(* IEC 61131-3 sources: SmartHomeNew/ (part 13) *)

(* ---- PRG_IO_Read_Phase_03_Environment_Sensors.st ---- *)
PROGRAM PRG_IO_Read_Phase_03_Environment_Sensors
VAR
    L_i : INT;
    L_Filtered_Room_Temp : REAL;
    L_Filtered_Floor_Temp : REAL;
    L_Any_Sensor_Fault : BOOL;

    fbCalib_Outdoor_Temp : FB_Sensor_Calibration_Processor;
    fbCalib_Supply_Temps : ARRAY[1..GVL_CONSTANTS.C_MAX_SUPPLY_TEMPS] OF FB_Sensor_Calibration_Processor;
    fbCalib_Room_Temps : ARRAY[1..GVL_CONSTANTS.C_MAX_ZONES] OF FB_Sensor_Calibration_Processor;
    fbCalib_Floor_Temps : ARRAY[1..GVL_CONSTANTS.C_MAX_ZONES] OF FB_Sensor_Calibration_Processor;
    fbCalib_Room_Hum : ARRAY[1..GVL_CONSTANTS.C_MAX_ZONES] OF FB_Sensor_Calibration_Processor;
    fbCalib_Room_CO2 : ARRAY[1..GVL_CONSTANTS.C_MAX_ZONES] OF FB_Sensor_Calibration_Processor;
END_VAR

L_Any_Sensor_Fault := FALSE;

fbCalib_Outdoor_Temp(
    VI_Raw_Value := GVL_IO.AI_Temp_Outdoor.rValue,
    VI_Record := GVL_CONFIG.G_Calib_Outdoor_Temp
);
GVL_STATE.G_Outdoor_Temp := fbCalib_Outdoor_Temp.VO_Calibrated_Value;

FOR L_i := 1 TO GVL_CONSTANTS.C_MAX_SUPPLY_TEMPS DO
    IF GVL_IO.AI_Supply_Temps[L_i].wStatus = 0 THEN
        fbCalib_Supply_Temps[L_i](
            VI_Raw_Value := GVL_IO.AI_Supply_Temps[L_i].rValue,
            VI_Record := GVL_CONFIG.G_Calib_Supply_Temps[L_i]
        );
        GVL_STATE.G_Supply_Temps[L_i] := fbCalib_Supply_Temps[L_i].VO_Calibrated_Value;
    ELSE
        L_Any_Sensor_Fault := TRUE;
    END_IF;
END_FOR;

FOR L_i := 1 TO GVL_CONSTANTS.C_MAX_ZONES DO
    fbCalib_Room_Hum[L_i](
        VI_Raw_Value := GVL_IO.AI_Room_Hum[L_i],
        VI_Record := GVL_CONFIG.G_Calib_Humidity[L_i]
    );
    GVL_STATE.G_Room_Hum[L_i] := fbCalib_Room_Hum[L_i].VO_Calibrated_Value;

    fbCalib_Room_CO2[L_i](
        VI_Raw_Value := GVL_IO.AI_Room_CO2[L_i],
        VI_Record := GVL_CONFIG.G_Calib_CO2[L_i]
    );
    GVL_STATE.G_Room_CO2[L_i] := fbCalib_Room_CO2[L_i].VO_Calibrated_Value;
END_FOR;

FOR L_i := 1 TO GVL_CONSTANTS.C_MAX_ZONES DO
    fbCalib_Room_Temps[L_i](
        VI_Raw_Value := GVL_IO.AI_Room_Temps[L_i],
        VI_Record := GVL_CONFIG.G_Calib_Room_Temps[L_i]
    );

    IF GVL_STATE.G_Last_Valid_Room_Temps[L_i] = 0.0 THEN
        L_Filtered_Room_Temp := fbCalib_Room_Temps[L_i].VO_Calibrated_Value;
    ELSE
        L_Filtered_Room_Temp := (GVL_STATE.G_Last_Valid_Room_Temps[L_i] * 0.9) + (fbCalib_Room_Temps[L_i].VO_Calibrated_Value * 0.1);
    END_IF;

    IF (L_Filtered_Room_Temp < -50.0) OR (L_Filtered_Room_Temp > 100.0) THEN
        GVL_STATE.G_Temp_Sensor_Fault[L_i] := TRUE;
        GVL_STATE.G_Room_Temps[L_i] := GVL_STATE.G_Last_Valid_Room_Temps[L_i];
        L_Any_Sensor_Fault := TRUE;
    ELSE
        GVL_STATE.G_Temp_Sensor_Fault[L_i] := FALSE;
        GVL_STATE.G_Room_Temps[L_i] := L_Filtered_Room_Temp;
        GVL_STATE.G_Last_Valid_Room_Temps[L_i] := L_Filtered_Room_Temp;
    END_IF;
END_FOR;

FOR L_i := 1 TO GVL_CONSTANTS.C_MAX_HEATING_CIRCUITS DO
    IF L_i <= GVL_CONSTANTS.C_MAX_ZONES THEN
        fbCalib_Floor_Temps[L_i](
            VI_Raw_Value := GVL_IO.AI_Floor_Temps[L_i],
            VI_Record := GVL_CONFIG.G_Calib_Floor_Temps[L_i]
        );

        IF GVL_STATE.G_Last_Valid_Floor_Temps[L_i] = 0.0 THEN
            L_Filtered_Floor_Temp := fbCalib_Floor_Temps[L_i].VO_Calibrated_Value;
        ELSE
            L_Filtered_Floor_Temp := (GVL_STATE.G_Last_Valid_Floor_Temps[L_i] * 0.9) + (fbCalib_Floor_Temps[L_i].VO_Calibrated_Value * 0.1);
        END_IF;

        IF (L_Filtered_Floor_Temp < -50.0) OR (L_Filtered_Floor_Temp > 100.0) THEN
            GVL_STATE.G_Floor_Temp_Sensor_Fault[L_i] := TRUE;
            GVL_STATE.G_Floor_Temps[L_i] := GVL_STATE.G_Last_Valid_Floor_Temps[L_i];
            L_Any_Sensor_Fault := TRUE;
        ELSE
            GVL_STATE.G_Floor_Temp_Sensor_Fault[L_i] := FALSE;
            GVL_STATE.G_Floor_Temps[L_i] := L_Filtered_Floor_Temp;
            GVL_STATE.G_Last_Valid_Floor_Temps[L_i] := L_Filtered_Floor_Temp;
        END_IF;
    ELSE
        GVL_STATE.G_Floor_Temp_Sensor_Fault[L_i] := TRUE;
        GVL_STATE.G_Floor_Temps[L_i] := GVL_STATE.G_Last_Valid_Floor_Temps[L_i];
        L_Any_Sensor_Fault := TRUE;
    END_IF;
END_FOR;

GVL_STATUS.G_Diagnostics.Sensor_Fault := L_Any_Sensor_Fault;

// >>> BULK_SYNC_ANCHOR: PRG_IO_Read_Phase_03_Environment_Sensors <<<
END_PROGRAM

(* ---- PRG_IO_Read_Phase_04_Heating_Manifold_Sensors.st ---- *)
PROGRAM PRG_IO_Read_Phase_04_Heating_Manifold_Sensors
VAR
    L_i : INT;
    L_Manifold_Pressure_Raw : WORD;
    L_Manifold_Current_Raw : WORD;

    fbDiagEventManager : FB_Diagnostics_Event_Manager;
    fbCalib_Manifold_T_Supply : ARRAY[1..GVL_CONSTANTS.C_MAX_MANIFOLDS] OF FB_Sensor_Calibration_Processor;
    fbCalib_Manifold_T_Return : ARRAY[1..GVL_CONSTANTS.C_MAX_MANIFOLDS] OF FB_Sensor_Calibration_Processor;
    fbAnalog_Manifold_Pressure : ARRAY[1..GVL_CONSTANTS.C_MAX_MANIFOLDS] OF FB_Sensor_Analog_Processing;
    fbAnalog_Manifold_Current : ARRAY[1..GVL_CONSTANTS.C_MAX_MANIFOLDS] OF FB_Sensor_Analog_Processing;
END_VAR

GVL_STATUS.G_Diagnostics.Manifold_Pressure_Fault_Active := FALSE;
GVL_STATUS.G_Diagnostics.Manifold_Pressure_First_Fault_Index := 0;
GVL_STATUS.G_Diagnostics.Manifold_Current_Fault_Active := FALSE;
GVL_STATUS.G_Diagnostics.Manifold_Current_First_Fault_Index := 0;
GVL_STATUS.G_Diagnostics.Manifold_Pressure_Fault_Text := '';
GVL_STATUS.G_Diagnostics.Manifold_Current_Fault_Text := '';

FOR L_i := 1 TO GVL_CONSTANTS.C_MAX_MANIFOLDS DO
    IF GVL_IO.AI_Manifold_Pressures[L_i] < 0 THEN
        L_Manifold_Pressure_Raw := 0;
    ELSE
        L_Manifold_Pressure_Raw := INT_TO_WORD(GVL_IO.AI_Manifold_Pressures[L_i]);
    END_IF;

    IF GVL_IO.AI_Manifold_Currents[L_i] < 0 THEN
        L_Manifold_Current_Raw := 0;
    ELSE
        L_Manifold_Current_Raw := INT_TO_WORD(GVL_IO.AI_Manifold_Currents[L_i]);
    END_IF;

    fbAnalog_Manifold_Pressure[L_i](
        VI_Raw_Value := L_Manifold_Pressure_Raw,
        VI_Sensor_Type := 0,
        VI_Min_Scale := 0.0,
        VI_Max_Scale := 10.0,
        VI_Offset := 0.0,
        VI_Multiplier := 1.0,
        VI_Filter_Time_MS := GVL_CONSTANTS.C_MS_IN_SECOND,
        VI_System_Time_MS := GVL_STATUS.G_System_Time_MS,
        VI_Fallback_Mode := 0,
        VI_Default_Value := 0.0
    );
    GVL_STATE.G_Manifold_Pressures[L_i] := fbAnalog_Manifold_Pressure[L_i].VO_Value;
    GVL_STATUS.G_Diagnostics.Manifold_Pressure_Fault[L_i] := fbAnalog_Manifold_Pressure[L_i].VO_Error;
    GVL_STATUS.G_Diagnostics.Manifold_Pressure_Diag_Code[L_i] := fbAnalog_Manifold_Pressure[L_i].VO_Diag_Code;

    fbDiagEventManager(
        VI_Code := GVL_CONFIG.ERR_PRESSURE_OUT_OF_RANGE,
        VI_Severity := 3,
        VI_Active := fbAnalog_Manifold_Pressure[L_i].VO_Error,
        VI_Timestamp := GVL_STATUS.G_System_Time_MS,
        VI_Source := 100 + L_i,
        VIO_Events := GVL_STATUS.G_Diagnostics_Events,
        VIO_Count := GVL_STATUS.G_Diagnostics_Count
    );

    fbAnalog_Manifold_Current[L_i](
        VI_Raw_Value := L_Manifold_Current_Raw,
        VI_Sensor_Type := 0,
        VI_Min_Scale := 0.0,
        VI_Max_Scale := 16.0,
        VI_Offset := 0.0,
        VI_Multiplier := 1.0,
        VI_Filter_Time_MS := GVL_CONSTANTS.C_MS_IN_SECOND,
        VI_System_Time_MS := GVL_STATUS.G_System_Time_MS,
        VI_Fallback_Mode := 0,
        VI_Default_Value := 0.0
    );
    GVL_STATE.G_Manifold_Currents[L_i] := fbAnalog_Manifold_Current[L_i].VO_Value;
    GVL_STATUS.G_Diagnostics.Manifold_Current_Fault[L_i] := fbAnalog_Manifold_Current[L_i].VO_Error;
    GVL_STATUS.G_Diagnostics.Manifold_Current_Diag_Code[L_i] := fbAnalog_Manifold_Current[L_i].VO_Diag_Code;

    fbDiagEventManager(
        VI_Code := GVL_CONFIG.ERR_PUMP_UNDERCURRENT,
        VI_Severity := 3,
        VI_Active := fbAnalog_Manifold_Current[L_i].VO_Error,
        VI_Timestamp := GVL_STATUS.G_System_Time_MS,
        VI_Source := 200 + L_i,
        VIO_Events := GVL_STATUS.G_Diagnostics_Events,
        VIO_Count := GVL_STATUS.G_Diagnostics_Count
    );

    IF GVL_IO.AI_Manifold_Temps_Supply[L_i].wStatus = 0 THEN
        fbCalib_Manifold_T_Supply[L_i](
            VI_Raw_Value := GVL_IO.AI_Manifold_Temps_Supply[L_i].rValue,
            VI_Record := GVL_CONFIG.G_Calib_Manifold_T_Supply[L_i]
        );
        GVL_STATE.G_Manifold_T_Supply[L_i] := fbCalib_Manifold_T_Supply[L_i].VO_Calibrated_Value;
    END_IF;

    fbCalib_Manifold_T_Return[L_i](
        VI_Raw_Value := INT_TO_REAL(GVL_IO.AI_Manifold_Temps_Return[L_i]) / 10.0,
        VI_Record := GVL_CONFIG.G_Calib_Manifold_T_Return[L_i]
    );
    GVL_STATE.G_Manifold_T_Return[L_i] := fbCalib_Manifold_T_Return[L_i].VO_Calibrated_Value;
    GVL_STATE.G_Manifold_End_Switches[L_i] := GVL_IO.DI_Manifold_End_Switches[L_i];

    IF GVL_STATUS.G_Diagnostics.Manifold_Pressure_Fault[L_i] OR GVL_STATUS.G_Diagnostics.Manifold_Current_Fault[L_i] THEN
        GVL_STATUS.G_Diagnostics.Sensor_Fault := TRUE;
        GVL_STATUS.G_Diagnostics.Subsystem_Degraded := TRUE;
    END_IF;

    IF GVL_STATUS.G_Diagnostics.Manifold_Pressure_Fault[L_i] AND GVL_STATUS.G_Diagnostics.Manifold_Current_Fault[L_i] THEN
        GVL_STATUS.G_Diagnostics.Manifold_Pressure_Fault_Text := 'Correlated pressure/current fault detected';
        GVL_STATUS.G_Diagnostics.Manifold_Current_Fault_Text := 'Correlated pressure/current fault detected';
    ELSIF GVL_STATUS.G_Diagnostics.Manifold_Pressure_Fault[L_i] AND (GVL_STATUS.G_Diagnostics.Manifold_Pressure_Fault_Text = '') THEN
        GVL_STATUS.G_Diagnostics.Manifold_Pressure_Fault_Text := 'Pressure sensor fault detected';
    ELSIF GVL_STATUS.G_Diagnostics.Manifold_Current_Fault[L_i] AND (GVL_STATUS.G_Diagnostics.Manifold_Current_Fault_Text = '') THEN
        GVL_STATUS.G_Diagnostics.Manifold_Current_Fault_Text := 'Current sensor fault detected';
    END_IF;
END_FOR;

// >>> BULK_SYNC_ANCHOR: PRG_IO_Read_Phase_04_Heating_Manifold_Sensors <<<
END_PROGRAM

(* ---- PRG_IO_Read_Phase_05_Gas_DHW_Water_Feedback.st ---- *)
PROGRAM PRG_IO_Read_Phase_05_Gas_DHW_Water_Feedback
VAR
    L_i : INT;

    fbDiagEventManager : FB_Diagnostics_Event_Manager;
    fbCalib_Methane : ARRAY[1..GVL_CONSTANTS.C_MAX_METHANE_SENSORS] OF FB_Sensor_Calibration_Processor;
    fbCalib_CO : ARRAY[1..GVL_CONSTANTS.C_MAX_CO_SENSORS] OF FB_Sensor_Calibration_Processor;
END_VAR

FOR L_i := 1 TO GVL_CONSTANTS.C_MAX_METHANE_SENSORS DO
    IF GVL_IO.AI_Methane_LEL[L_i].wStatus = 0 THEN
        fbCalib_Methane[L_i](
            VI_Raw_Value := GVL_IO.AI_Methane_LEL[L_i].rValue,
            VI_Record := GVL_CONFIG.G_Calib_Methane[L_i]
        );
        GVL_STATE.G_Methane_Sensors[L_i] := fbCalib_Methane[L_i].VO_Calibrated_Value;
    END_IF;

    fbDiagEventManager(
        VI_Code := 16#E003,
        VI_Severity := 3,
        VI_Active := GVL_IO.AI_Methane_LEL[L_i].wStatus <> 0,
        VI_Timestamp := GVL_STATUS.G_System_Time_MS,
        VI_Source := 300 + L_i,
        VIO_Events := GVL_STATUS.G_Diagnostics_Events,
        VIO_Count := GVL_STATUS.G_Diagnostics_Count
    );
END_FOR;

FOR L_i := 1 TO GVL_CONSTANTS.C_MAX_CO_SENSORS DO
    fbCalib_CO[L_i](
        VI_Raw_Value := GVL_IO.AI_CO_PPM[L_i],
        VI_Record := GVL_CONFIG.G_Calib_CO[L_i]
    );
    GVL_STATE.G_CO_Sensors[L_i] := fbCalib_CO[L_i].VO_Calibrated_Value;
END_FOR;

GVL_STATE.G_DHW_Temp := GVL_IO.AI_DHW_Temp;
GVL_STATE.G_DHW_Pressure := GVL_IO.AI_DHW_Pressure;

GVL_STATE.G_Water_Zone_Open_FB := GVL_IO.DI_Water_Zone_Open_FB;
GVL_STATE.G_Water_Zone_Close_FB := GVL_IO.DI_Water_Zone_Close_FB;

// >>> BULK_SYNC_ANCHOR: PRG_IO_Read_Phase_05_Gas_DHW_Water_Feedback <<<
END_PROGRAM

(* ---- PRG_IO_Write.st ---- *)
PROGRAM PRG_IO_Write
VAR
    L_i : INT;
    L_Heating_Forced_Off : BOOL;
    L_Vent_Forced_Off : BOOL;
    L_Water_Forced_Off : BOOL;
    L_Access_Forced_Off : BOOL;
    L_Access_Safety_Override : BOOL;
    L_Global_Hard_Stop : BOOL;
    L_Gas_Safety_Stop : BOOL;
    L_Freeze_Active : BOOL;
    L_Gas_Fire_Siren_Enable : BOOL;
    L_PreOutput_Block_IO : BOOL;
    L_Output_Freshness_Block : BOOL;
    L_Snapshot_Block : BOOL;
    L_Distributed_Execution_Block : BOOL;
    L_Gas_Siren_Authority : BOOL;
    L_Fire_Siren_Authority : BOOL;
    fbTrace : FB_Trace_Write;
END_VAR

L_PreOutput_Block_IO := GVL_COMMAND_VERIFY.PreOutput_Block_IO;
L_Output_Freshness_Block := GVL_OUTPUT_EPOCH.Output_Forced_Safe_Decay;
L_Snapshot_Block := (NOT GVL_RUNTIME_SNAPSHOT.Snapshot_Frozen) OR (NOT GVL_RUNTIME_SNAPSHOT.Snapshot_Publication_Allowed) OR (NOT GVL_RUNTIME_SNAPSHOT.Snapshot_Copy_Valid) OR (NOT GVL_RUNTIME_SNAPSHOT.Snapshot_Isolation_Valid) OR GVL_RUNTIME_SNAPSHOT.Snapshot_Mutation_Detected;

L_Distributed_Execution_Block :=
    NOT GVL_Distributed_Execution_Gates.G_Can_Execute
    OR NOT GVL_Distributed_Execution_Gates.G_Can_Own_Projection;

L_Global_Hard_Stop :=
    GVL_COMMAND_SHADOW.G_Heating_Emergency_Stop
    OR L_PreOutput_Block_IO
    OR L_Output_Freshness_Block
    OR L_Snapshot_Block
    OR L_Distributed_Execution_Block;

L_Gas_Safety_Stop := GVL_COMMAND_SHADOW.G_Heating_Gas_Safety_Stop OR GVL_COMMAND_SHADOW.G_Boiler_Stop;
L_Freeze_Active := GVL_STATE.G_Safety_Freeze_Risk;
L_Gas_Fire_Siren_Enable := GVL_ALARM.G_Gas_Fire_Siren OR GVL_ALARM.G_Global_Siren OR GVL_ALARM.G_Global_Critical;

// Physical siren actuation must use authoritative safety truth,
// not stale alarm projection fields.
L_Gas_Siren_Authority := GVL_HEALTH_BRIDGE.G_Gas_Detected OR GVL_HEALTH_BRIDGE.G_CO_Alarm_Level OR GVL_STATE.G_Safety_Gas_Latched;
L_Fire_Siren_Authority := GVL_HEALTH_BRIDGE.G_Smoke_Detected OR GVL_STATE.G_Safety_Smoke_Latched;

// ======================================================
// AUTHORITATIVE IO HARD-STOP GATE
// ======================================================
// Physical IO publication must never continue when:
//   - PLC authority is lost;
//   - distributed execution gates restricted execution;
//   - emergency stop is active;
//   - pre-output barrier rejected current-cycle runtime projection;
//   - output freshness governor invalidated publication;
//   - immutable snapshot authority invalidated publication;
//   - snapshot mutation was detected.
// ======================================================

IF NOT GVL_STATUS.G_Is_Active_PLC OR L_Global_Hard_Stop THEN
    FOR L_i := 1 TO GVL_CONSTANTS.C_MAX_HEATING_CIRCUITS DO
        GVL_IO.DO_Zone_Valves[L_i] := FALSE;
    END_FOR;

    FOR L_i := 1 TO GVL_CONSTANTS.C_MAX_MANIFOLDS DO
        GVL_IO.DO_Manifold_Pumps[L_i] := FALSE;
        GVL_IO.AO_Manifold_Valves[L_i] := 0;
    END_FOR;

    GVL_IO.DO_DHW_Heating_Pump := FALSE;
    GVL_IO.DO_DHW_Circ_Pump := FALSE;
    GVL_IO.DO_Backup_Circulation_Pump := FALSE;
    GVL_IO.DO_Electric_Heater_Enable := FALSE;

    FOR L_i := 1 TO GVL_CONSTANTS.C_MAX_SUPPLY_FANS DO
        GVL_IO.AO_Supply_Fans[L_i] := 0;
    END_FOR;

    FOR L_i := 1 TO GVL_CONSTANTS.C_MAX_EXHAUST_FANS DO
        GVL_IO.AO_Exhaust_Fans[L_i] := 0;
    END_FOR;

    FOR L_i := 1 TO GVL_CONSTANTS.C_MAX_WATER_ZONES DO
        GVL_IO.DO_Water_Zone_Enable[L_i] := FALSE;
    END_FOR;

    FOR L_i := 1 TO GVL_CONSTANTS.C_MAX_LIGHT_ZONES DO
        GVL_IO.AO_Lighting_Levels[L_i] := 0;
    END_FOR;

    FOR L_i := 1 TO GVL_CONSTANTS.C_MAX_BLINDS DO
        GVL_IO.AO_Blinds_Positions[L_i] := 1000;
    END_FOR;

    FOR L_i := 1 TO GVL_CONSTANTS.C_MAX_SOCKETS DO
        GVL_IO.DO_Sockets[L_i] := FALSE;
    END_FOR;

    GVL_IO.DO_Gate_Open := FALSE;
    GVL_IO.DO_Wicket_Open := FALSE;
    GVL_IO.DO_Lock_1_Open := FALSE;
    GVL_IO.DO_Lock_1_Close := FALSE;
    GVL_IO.DO_Lock_2_Open := FALSE;
    GVL_IO.DO_Lock_2_Close := FALSE;
    GVL_IO.DO_Gas_Siren := L_Gas_Fire_Siren_Enable AND L_Gas_Siren_Authority;
    GVL_IO.DO_Fire_Siren := L_Gas_Fire_Siren_Enable AND L_Fire_Siren_Authority;
    GVL_IO.DO_Security_Siren := GVL_ALARM.G_Security_Siren OR (GVL_ALARM.G_Global_Siren AND GVL_ALARM.G_Security_Alarm);
    GVL_IO.DO_Gas_Valve_Close := TRUE;

    IF L_Distributed_Execution_Block THEN
        fbTrace(iLayer := TRACE_IO,iSource := SRC_IO,iReason := REASON_SAFETY_BLOCK,iValueBool := TRUE,iValueReal := 999.0,iText := 'IO blocked by distributed execution governance');
    END_IF;

    IF L_PreOutput_Block_IO THEN
        fbTrace(iLayer := TRACE_IO,iSource := SRC_IO,iReason := REASON_SAFETY_BLOCK,iValueBool := TRUE,iValueReal := UDINT_TO_REAL(GVL_COMMAND_VERIFY.PreOutput_Last_Error_Code),iText := 'IO blocked by pre-output barrier');
    END_IF;

    IF L_Output_Freshness_Block THEN
        fbTrace(iLayer := TRACE_IO,iSource := SRC_IO,iReason := REASON_SAFETY_BLOCK,iValueBool := TRUE,iValueReal := UDINT_TO_REAL(GVL_OUTPUT_EPOCH.Output_Last_Error_Code),iText := 'IO forced safe by output freshness decay');
    END_IF;

    IF L_Snapshot_Block THEN
        fbTrace(iLayer := TRACE_IO,iSource := SRC_IO,iReason := REASON_SAFETY_BLOCK,iValueBool := TRUE,iValueReal := UDINT_TO_REAL(GVL_RUNTIME_SNAPSHOT.Snapshot_Last_Error_Code),iText := 'IO blocked by immutable snapshot authority');
    END_IF;

    RETURN;
END_IF;

L_Heating_Forced_Off := GVL_COMMAND_SHADOW.G_Heating_Block;
L_Vent_Forced_Off := GVL_COMMAND_SHADOW.G_Vent_Stop OR GVL_COMMAND_SHADOW.G_Vent_Block;
L_Water_Forced_Off := GVL_COMMAND_SHADOW.G_Water_Block OR GVL_COMMAND_SHADOW.G_Water_Emergency_Stop;

L_Access_Safety_Override := (GVL_SAFETY_SHUTDOWN.G_Safety_Mode = FIRE) OR (GVL_SAFETY_SHUTDOWN.G_Safety_Mode = GAS);
L_Access_Forced_Off := GVL_SAFETY_RECOVERY.G_Recovery_Active AND NOT L_Access_Safety_Override;

FOR L_i := 1 TO GVL_CONSTANTS.C_MAX_HEATING_CIRCUITS DO
    IF (L_i > GVL_SYSTEM_SIZE_CONFIG.G_Active_Heating_Circuits) OR L_Heating_Forced_Off THEN
        GVL_IO.DO_Zone_Valves[L_i] := FALSE;
    ELSE
        GVL_IO.DO_Zone_Valves[L_i] := GVL_HEATING_OUTPUT.DO_Zone_Valves[L_i];
    END_IF;
END_FOR;

FOR L_i := 1 TO GVL_CONSTANTS.C_MAX_MANIFOLDS DO
    IF L_Heating_Forced_Off AND NOT (L_Gas_Safety_Stop AND L_Freeze_Active) THEN
        GVL_IO.DO_Manifold_Pumps[L_i] := FALSE;
        GVL_IO.AO_Manifold_Valves[L_i] := 0;
    ELSE
        GVL_IO.DO_Manifold_Pumps[L_i] := GVL_HEATING_OUTPUT.DO_Manifold_Pumps[L_i];
        GVL_IO.AO_Manifold_Valves[L_i] := GVL_HEATING_OUTPUT.AO_Manifold_Valves[L_i];
    END_IF;
END_FOR;

IF L_Heating_Forced_Off AND NOT (L_Gas_Safety_Stop AND L_Freeze_Active) THEN
    GVL_IO.DO_DHW_Heating_Pump := FALSE;
    GVL_IO.DO_DHW_Circ_Pump := FALSE;
    GVL_IO.DO_Backup_Circulation_Pump := FALSE;
    GVL_IO.DO_Electric_Heater_Enable := FALSE;
ELSE
    GVL_IO.DO_DHW_Heating_Pump := GVL_HEATING_OUTPUT.DO_DHW_Heating_Pump;
    GVL_IO.DO_DHW_Circ_Pump := GVL_HEATING_OUTPUT.DO_DHW_Circ_Pump;
    GVL_IO.DO_Backup_Circulation_Pump := GVL_HEATING_OUTPUT.DO_Backup_Circulation_Pump;
    GVL_IO.DO_Electric_Heater_Enable := GVL_HEATING_OUTPUT.DO_Electric_Heater_Enable;
END_IF;

FOR L_i := 1 TO GVL_CONSTANTS.C_MAX_SUPPLY_FANS DO
    IF L_Vent_Forced_Off THEN
        GVL_IO.AO_Supply_Fans[L_i] := 0;
    ELSE
        GVL_IO.AO_Supply_Fans[L_i] := GVL_VENT_OUTPUT.AO_Supply_Fans[L_i];
    END_IF;
END_FOR;

FOR L_i := 1 TO GVL_CONSTANTS.C_MAX_EXHAUST_FANS DO
    IF L_Vent_Forced_Off THEN
        GVL_IO.AO_Exhaust_Fans[L_i] := 0;
    ELSE
        GVL_IO.AO_Exhaust_Fans[L_i] := GVL_VENT_OUTPUT.AO_Exhaust_Fans[L_i];
    END_IF;
END_FOR;

GVL_IO.DO_Water_Valve_35_Close := GVL_WATER_OUTPUT.DO_Water_Valve_35_Close;
GVL_IO.DO_Water_Valve_36_Close := GVL_WATER_OUTPUT.DO_Water_Valve_36_Close;

FOR L_i := 1 TO GVL_CONSTANTS.C_MAX_WATER_ZONES DO
    IF (L_i > GVL_SYSTEM_SIZE_CONFIG.G_Active_Water_Zones) OR L_Water_Forced_Off THEN
        GVL_IO.DO_Water_Zone_Enable[L_i] := FALSE;
    ELSE
        GVL_IO.DO_Water_Zone_Enable[L_i] := GVL_WATER_OUTPUT.DO_Water_Zone_Enable[L_i];
    END_IF;
END_FOR;

FOR L_i := 1 TO GVL_CONSTANTS.C_MAX_LIGHT_ZONES DO
    GVL_IO.AO_Lighting_Levels[L_i] := GVL_LIGHTING_OUTPUT.AO_Lighting_Levels[L_i];
END_FOR;

FOR L_i := 1 TO GVL_CONSTANTS.C_MAX_BLINDS DO
    GVL_IO.AO_Blinds_Positions[L_i] := GVL_LIGHTING_OUTPUT.AO_Blinds_Positions[L_i];
END_FOR;

FOR L_i := 1 TO GVL_CONSTANTS.C_MAX_SOCKETS DO
    GVL_IO.DO_Sockets[L_i] := GVL_LIGHTING_OUTPUT.DO_Sockets[L_i];
END_FOR;

IF L_Access_Forced_Off THEN
    GVL_IO.DO_Gate_Open := FALSE;
    GVL_IO.DO_Wicket_Open := FALSE;
    GVL_IO.DO_Lock_1_Open := FALSE;
    GVL_IO.DO_Lock_1_Close := FALSE;
    GVL_IO.DO_Lock_2_Open := FALSE;
    GVL_IO.DO_Lock_2_Close := FALSE;
ELSE
    GVL_IO.DO_Gate_Open := GVL_ACCESS_OUTPUT.DO_Gate_Open;
    GVL_IO.DO_Wicket_Open := GVL_ACCESS_OUTPUT.DO_Wicket_Open;
    GVL_IO.DO_Lock_1_Open := GVL_ACCESS_OUTPUT.DO_Lock_1_Open;
    GVL_IO.DO_Lock_1_Close := GVL_ACCESS_OUTPUT.DO_Lock_1_Close;
    GVL_IO.DO_Lock_2_Open := GVL_ACCESS_OUTPUT.DO_Lock_2_Open;
    GVL_IO.DO_Lock_2_Close := GVL_ACCESS_OUTPUT.DO_Lock_2_Close;
END_IF;

GVL_IO.DO_Gas_Siren := L_Gas_Fire_Siren_Enable AND L_Gas_Siren_Authority;
GVL_IO.DO_Fire_Siren := L_Gas_Fire_Siren_Enable AND L_Fire_Siren_Authority;
GVL_IO.DO_Security_Siren := GVL_ALARM.G_Security_Siren OR (GVL_ALARM.G_Global_Siren AND GVL_ALARM.G_Security_Alarm);
GVL_IO.DO_Gas_Valve_Close := GVL_COMMAND_SHADOW.G_Gas_Valve_Close;

fbTrace(iLayer := TRACE_IO,iSource := SRC_IO,iReason := REASON_DOMAIN_PROJECTION,iValueBool := TRUE,iValueReal := 0.0,iText := 'IO write projection executed');
END_PROGRAM

(* ---- PRG_IO_Write_Phase_01_Context.st ---- *)
PROGRAM PRG_IO_Write_Phase_01_Context

GVL_IO_WRITE_RUNTIME_BUFFER.B_PreOutput_Block_IO :=
    GVL_COMMAND_VERIFY.PreOutput_Block_IO;

GVL_IO_WRITE_RUNTIME_BUFFER.B_Output_Freshness_Block :=
    GVL_OUTPUT_EPOCH.Output_Forced_Safe_Decay;

GVL_IO_WRITE_RUNTIME_BUFFER.B_Output_Publication_Block :=
    (NOT GVL_OUTPUT_EPOCH.Output_Publication_Valid)
    OR (NOT GVL_OUTPUT_EPOCH.Output_Runtime_Epoch_Valid)
    OR GVL_OUTPUT_EPOCH.Output_Lease_Expired;

GVL_IO_WRITE_RUNTIME_BUFFER.B_Distributed_Publication_Block :=
    (NOT GVL_DISTRIBUTED_COMMIT.Distributed_Commit_Valid)
    OR GVL_DISTRIBUTED_COMMIT.Distributed_Commit_Quarantine_Active
    OR GVL_DISTRIBUTED_COMMIT.Commit_Lease_Expired
    OR (NOT GVL_DISTRIBUTED_SNAPSHOT.Distributed_Publication_Reconciled)
    OR (NOT GVL_DISTRIBUTED_SNAPSHOT.Distributed_Publication_Freeze_Valid)
    OR (NOT GVL_DISTRIBUTED_SNAPSHOT.Distributed_Snapshot_Consistent);

GVL_IO_WRITE_RUNTIME_BUFFER.B_Snapshot_Block :=
    (NOT GVL_RUNTIME_SNAPSHOT.Snapshot_Frozen)
    OR (NOT GVL_RUNTIME_SNAPSHOT.Snapshot_Publication_Allowed)
    OR (NOT GVL_RUNTIME_SNAPSHOT.Snapshot_Copy_Valid)
    OR (NOT GVL_RUNTIME_SNAPSHOT.Snapshot_Isolation_Valid)
    OR GVL_RUNTIME_SNAPSHOT.Snapshot_Mutation_Detected;

GVL_IO_WRITE_RUNTIME_BUFFER.B_Distributed_Execution_Block :=
    NOT GVL_Distributed_Execution_Gates.G_Can_Execute
    OR NOT GVL_Distributed_Execution_Gates.G_Can_Own_Projection;

GVL_IO_WRITE_RUNTIME_BUFFER.B_Global_Hard_Stop :=
    (GVL_SAFETY_SHUTDOWN.G_Safety_Mode = GLOBAL_STOP)
    OR GVL_IO_WRITE_RUNTIME_BUFFER.B_PreOutput_Block_IO
    OR GVL_IO_WRITE_RUNTIME_BUFFER.B_Output_Freshness_Block
    OR GVL_IO_WRITE_RUNTIME_BUFFER.B_Output_Publication_Block
    OR GVL_IO_WRITE_RUNTIME_BUFFER.B_Distributed_Publication_Block
    OR GVL_IO_WRITE_RUNTIME_BUFFER.B_Snapshot_Block
    OR GVL_IO_WRITE_RUNTIME_BUFFER.B_Distributed_Execution_Block;

GVL_IO_WRITE_RUNTIME_BUFFER.B_Gas_Safety_Stop :=
    GVL_COMMAND_SHADOW.G_Heating_Gas_Safety_Stop
    OR GVL_COMMAND_SHADOW.G_Boiler_Stop;

GVL_IO_WRITE_RUNTIME_BUFFER.B_Freeze_Active :=
    GVL_STATE.G_Safety_Freeze_Risk;

GVL_IO_WRITE_RUNTIME_BUFFER.B_Gas_Fire_Siren_Enable :=
    GVL_ALARM.G_Gas_Fire_Siren
    OR GVL_ALARM.G_Global_Siren
    OR GVL_ALARM.G_Global_Critical;

GVL_IO_WRITE_RUNTIME_BUFFER.B_Gas_Siren_Authority :=
    GVL_HEALTH_BRIDGE.G_Gas_Detected
    OR GVL_HEALTH_BRIDGE.G_CO_Alarm_Level
    OR GVL_STATE.G_Safety_Gas_Latched;

GVL_IO_WRITE_RUNTIME_BUFFER.B_Fire_Siren_Authority :=
    GVL_HEALTH_BRIDGE.G_Smoke_Detected
    OR GVL_STATE.G_Safety_Smoke_Latched;

GVL_IO_WRITE_RUNTIME_BUFFER.B_Heating_Forced_Off :=
    GVL_COMMAND_SHADOW.G_Heating_Block
    OR GVL_COMMAND_SHADOW.G_Heating_Emergency_Stop;

GVL_IO_WRITE_RUNTIME_BUFFER.B_Vent_Forced_Off :=
    GVL_COMMAND_SHADOW.G_Vent_Stop
    OR GVL_COMMAND_SHADOW.G_Vent_Block;

GVL_IO_WRITE_RUNTIME_BUFFER.B_Water_Forced_Off :=
    GVL_COMMAND_SHADOW.G_Water_Block
    OR GVL_COMMAND_SHADOW.G_Water_Emergency_Stop;

GVL_IO_WRITE_RUNTIME_BUFFER.B_Access_Safety_Override :=
    (GVL_SAFETY_SHUTDOWN.G_Safety_Mode = FIRE)
    OR (GVL_SAFETY_SHUTDOWN.G_Safety_Mode = GAS);

GVL_IO_WRITE_RUNTIME_BUFFER.B_Access_Forced_Off :=
    GVL_SAFETY_RECOVERY.G_Recovery_Active
    AND NOT GVL_IO_WRITE_RUNTIME_BUFFER.B_Access_Safety_Override;

// >>> BULK_SYNC_ANCHOR: PRG_IO_Write_Phase_01_Context <<<
END_PROGRAM

(* ---- PRG_IO_Write_Phase_02_Hard_Stop_Safe_State.st ---- *)
PROGRAM PRG_IO_Write_Phase_02_Hard_Stop_Safe_State
// IO write phase 02: publish hard-stop safe physical outputs.
VAR
    L_i : INT;
    fbTrace : FB_Trace_Write;
END_VAR

FOR L_i := 1 TO GVL_CONSTANTS.C_MAX_HEATING_CIRCUITS DO
    GVL_IO.DO_Zone_Valves[L_i] := FALSE;
END_FOR;

FOR L_i := 1 TO GVL_CONSTANTS.C_MAX_MANIFOLDS DO
    GVL_IO.DO_Manifold_Pumps[L_i] := FALSE;
    GVL_IO.AO_Manifold_Valves[L_i] := 0;
END_FOR;

GVL_IO.DO_DHW_Heating_Pump := FALSE;
GVL_IO.DO_DHW_Circ_Pump := FALSE;
GVL_IO.DO_Backup_Circulation_Pump := FALSE;
GVL_IO.DO_Electric_Heater_Enable := FALSE;

FOR L_i := 1 TO GVL_CONSTANTS.C_MAX_SUPPLY_FANS DO
    GVL_IO.AO_Supply_Fans[L_i] := 0;
END_FOR;

FOR L_i := 1 TO GVL_CONSTANTS.C_MAX_EXHAUST_FANS DO
    GVL_IO.AO_Exhaust_Fans[L_i] := 0;
END_FOR;

FOR L_i := 1 TO GVL_CONSTANTS.C_MAX_WATER_ZONES DO
    GVL_IO.DO_Water_Zone_Enable[L_i] := FALSE;
END_FOR;

FOR L_i := 1 TO GVL_CONSTANTS.C_MAX_LIGHT_ZONES DO
    GVL_IO.AO_Lighting_Levels[L_i] := 0;
END_FOR;

FOR L_i := 1 TO GVL_CONSTANTS.C_MAX_BLINDS DO
    GVL_IO.AO_Blinds_Positions[L_i] := 1000;
END_FOR;

FOR L_i := 1 TO GVL_CONSTANTS.C_MAX_SOCKETS DO
    GVL_IO.DO_Sockets[L_i] := FALSE;
END_FOR;

GVL_IO.DO_Gate_Open := FALSE;
GVL_IO.DO_Wicket_Open := FALSE;
GVL_IO.DO_Lock_1_Open := FALSE;
GVL_IO.DO_Lock_1_Close := FALSE;
GVL_IO.DO_Lock_2_Open := FALSE;
GVL_IO.DO_Lock_2_Close := FALSE;

GVL_IO.DO_Water_Valve_35_Close := TRUE;
GVL_IO.DO_Water_Valve_36_Close := TRUE;
GVL_IO.DO_Gas_Valve_Close := TRUE;

GVL_IO.DO_Gas_Siren :=
    GVL_IO_WRITE_RUNTIME_BUFFER.B_Gas_Fire_Siren_Enable
    AND GVL_IO_WRITE_RUNTIME_BUFFER.B_Gas_Siren_Authority;

GVL_IO.DO_Fire_Siren :=
    GVL_IO_WRITE_RUNTIME_BUFFER.B_Gas_Fire_Siren_Enable
    AND GVL_IO_WRITE_RUNTIME_BUFFER.B_Fire_Siren_Authority;

GVL_IO.DO_Security_Siren :=
    GVL_ALARM.G_Security_Siren
    OR (GVL_ALARM.G_Global_Siren AND GVL_ALARM.G_Security_Alarm);

IF GVL_IO_WRITE_RUNTIME_BUFFER.B_Distributed_Publication_Block THEN
    fbTrace(
        iLayer := TRACE_IO,
        iSource := SRC_IO,
        iReason := REASON_SAFETY_BLOCK,
        iValueBool := TRUE,
        iValueReal := UDINT_TO_REAL(GVL_DISTRIBUTED_COMMIT.Distributed_Commit_Last_Error_Code),
        iText := 'IO blocked by distributed publication continuity authority'
    );
END_IF;

IF GVL_IO_WRITE_RUNTIME_BUFFER.B_Output_Publication_Block THEN
    fbTrace(
        iLayer := TRACE_IO,
        iSource := SRC_IO,
        iReason := REASON_SAFETY_BLOCK,
        iValueBool := TRUE,
        iValueReal := UDINT_TO_REAL(GVL_OUTPUT_EPOCH.Output_Last_Error_Code),
        iText := 'IO blocked by finalized output publication authority'
    );
END_IF;

// >>> BULK_SYNC_ANCHOR: PRG_IO_Write_Phase_02_Hard_Stop_Safe_State <<<
END_PROGRAM

(* ---- PRG_IO_Write_Phase_03_Domain_Projection.st ---- *)
PROGRAM PRG_IO_Write_Phase_03_Domain_Projection
// IO write phase 03: publish normal domain output projections.
VAR
    L_i : INT;
END_VAR

FOR L_i := 1 TO GVL_CONSTANTS.C_MAX_HEATING_CIRCUITS DO
    IF (L_i > GVL_SYSTEM_SIZE_CONFIG.G_Active_Heating_Circuits)
       OR GVL_IO_WRITE_RUNTIME_BUFFER.B_Heating_Forced_Off THEN
        GVL_IO.DO_Zone_Valves[L_i] := FALSE;
    ELSE
        GVL_IO.DO_Zone_Valves[L_i] := GVL_HEATING_OUTPUT.DO_Zone_Valves[L_i];
    END_IF;
END_FOR;

FOR L_i := 1 TO GVL_CONSTANTS.C_MAX_MANIFOLDS DO
    IF GVL_IO_WRITE_RUNTIME_BUFFER.B_Heating_Forced_Off
       AND NOT (GVL_IO_WRITE_RUNTIME_BUFFER.B_Gas_Safety_Stop
                AND GVL_IO_WRITE_RUNTIME_BUFFER.B_Freeze_Active) THEN
        GVL_IO.DO_Manifold_Pumps[L_i] := FALSE;
        GVL_IO.AO_Manifold_Valves[L_i] := 0;
    ELSE
        GVL_IO.DO_Manifold_Pumps[L_i] := GVL_HEATING_OUTPUT.DO_Manifold_Pumps[L_i];
        GVL_IO.AO_Manifold_Valves[L_i] := GVL_HEATING_OUTPUT.AO_Manifold_Valves[L_i];
    END_IF;
END_FOR;

IF GVL_IO_WRITE_RUNTIME_BUFFER.B_Heating_Forced_Off
   AND NOT (GVL_IO_WRITE_RUNTIME_BUFFER.B_Gas_Safety_Stop
            AND GVL_IO_WRITE_RUNTIME_BUFFER.B_Freeze_Active) THEN
    GVL_IO.DO_DHW_Heating_Pump := FALSE;
    GVL_IO.DO_DHW_Circ_Pump := FALSE;
    GVL_IO.DO_Backup_Circulation_Pump := FALSE;
    GVL_IO.DO_Electric_Heater_Enable := FALSE;
ELSE
    GVL_IO.DO_DHW_Heating_Pump := GVL_HEATING_OUTPUT.DO_DHW_Heating_Pump;
    GVL_IO.DO_DHW_Circ_Pump := GVL_HEATING_OUTPUT.DO_DHW_Circ_Pump;
    GVL_IO.DO_Backup_Circulation_Pump := GVL_HEATING_OUTPUT.DO_Backup_Circulation_Pump;
    GVL_IO.DO_Electric_Heater_Enable := GVL_HEATING_OUTPUT.DO_Electric_Heater_Enable;
END_IF;

FOR L_i := 1 TO GVL_CONSTANTS.C_MAX_SUPPLY_FANS DO
    IF GVL_IO_WRITE_RUNTIME_BUFFER.B_Vent_Forced_Off THEN
        GVL_IO.AO_Supply_Fans[L_i] := 0;
    ELSE
        GVL_IO.AO_Supply_Fans[L_i] := GVL_VENT_OUTPUT.AO_Supply_Fans[L_i];
    END_IF;
END_FOR;

FOR L_i := 1 TO GVL_CONSTANTS.C_MAX_EXHAUST_FANS DO
    IF GVL_IO_WRITE_RUNTIME_BUFFER.B_Vent_Forced_Off THEN
        GVL_IO.AO_Exhaust_Fans[L_i] := 0;
    ELSE
        GVL_IO.AO_Exhaust_Fans[L_i] := GVL_VENT_OUTPUT.AO_Exhaust_Fans[L_i];
    END_IF;
END_FOR;

GVL_IO.DO_Water_Valve_35_Close :=
    GVL_WATER_OUTPUT.DO_Water_Valve_35_Close
    OR GVL_COMMAND_SHADOW.G_Close_Valve_35;

GVL_IO.DO_Water_Valve_36_Close :=
    GVL_WATER_OUTPUT.DO_Water_Valve_36_Close
    OR GVL_COMMAND_SHADOW.G_Close_Valve_36;

FOR L_i := 1 TO GVL_CONSTANTS.C_MAX_WATER_ZONES DO
    IF (L_i > GVL_SYSTEM_SIZE_CONFIG.G_Active_Water_Zones)
       OR GVL_IO_WRITE_RUNTIME_BUFFER.B_Water_Forced_Off THEN
        GVL_IO.DO_Water_Zone_Enable[L_i] := FALSE;
    ELSE
        GVL_IO.DO_Water_Zone_Enable[L_i] := GVL_WATER_OUTPUT.DO_Water_Zone_Enable[L_i];
    END_IF;
END_FOR;

FOR L_i := 1 TO GVL_CONSTANTS.C_MAX_LIGHT_ZONES DO
    IF L_i > GVL_SYSTEM_SIZE_CONFIG.G_Active_Light_Zones THEN
        GVL_IO.AO_Lighting_Levels[L_i] := 0;
    ELSE
        GVL_IO.AO_Lighting_Levels[L_i] := GVL_LIGHTING_OUTPUT.AO_Lighting_Levels[L_i];
    END_IF;
END_FOR;

FOR L_i := 1 TO GVL_CONSTANTS.C_MAX_BLINDS DO
    IF L_i > GVL_SYSTEM_SIZE_CONFIG.G_Active_Blinds THEN
        GVL_IO.AO_Blinds_Positions[L_i] := 1000;
    ELSE
        GVL_IO.AO_Blinds_Positions[L_i] := GVL_LIGHTING_OUTPUT.AO_Blinds_Positions[L_i];
    END_IF;
END_FOR;

FOR L_i := 1 TO GVL_CONSTANTS.C_MAX_SOCKETS DO
    IF L_i > GVL_SYSTEM_SIZE_CONFIG.G_Active_Sockets THEN
        GVL_IO.DO_Sockets[L_i] := FALSE;
    ELSE
        GVL_IO.DO_Sockets[L_i] := GVL_LIGHTING_OUTPUT.DO_Sockets[L_i];
    END_IF;
END_FOR;

IF GVL_IO_WRITE_RUNTIME_BUFFER.B_Access_Forced_Off THEN
    GVL_IO.DO_Gate_Open := FALSE;
    GVL_IO.DO_Wicket_Open := FALSE;
    GVL_IO.DO_Lock_1_Open := FALSE;
    GVL_IO.DO_Lock_1_Close := FALSE;
    GVL_IO.DO_Lock_2_Open := FALSE;
    GVL_IO.DO_Lock_2_Close := FALSE;
ELSE
    GVL_IO.DO_Gate_Open := GVL_ACCESS_OUTPUT.DO_Gate_Open;
    GVL_IO.DO_Wicket_Open := GVL_ACCESS_OUTPUT.DO_Wicket_Open;
    GVL_IO.DO_Lock_1_Open := GVL_ACCESS_OUTPUT.DO_Lock_1_Open;
    GVL_IO.DO_Lock_1_Close := GVL_ACCESS_OUTPUT.DO_Lock_1_Close;
    GVL_IO.DO_Lock_2_Open := GVL_ACCESS_OUTPUT.DO_Lock_2_Open;
    GVL_IO.DO_Lock_2_Close := GVL_ACCESS_OUTPUT.DO_Lock_2_Close;
END_IF;

// >>> BULK_SYNC_ANCHOR: PRG_IO_Write_Phase_03_Domain_Projection <<<
END_PROGRAM

(* ---- PRG_IO_Write_Phase_04_Alarm_Trace.st ---- *)
PROGRAM PRG_IO_Write_Phase_04_Alarm_Trace
// IO write phase 04: publish final sirens, gas valve and normal trace.
VAR
    fbTrace : FB_Trace_Write;
    L_Audible_Siren_Allowed : BOOL;
END_VAR

L_Audible_Siren_Allowed := NOT GVL_ALARM_AUDIBLE_ACK.G_Ack_Active;

GVL_IO.DO_Gas_Siren :=
    L_Audible_Siren_Allowed
    AND GVL_IO_WRITE_RUNTIME_BUFFER.B_Gas_Fire_Siren_Enable
    AND GVL_IO_WRITE_RUNTIME_BUFFER.B_Gas_Siren_Authority;

GVL_IO.DO_Fire_Siren :=
    L_Audible_Siren_Allowed
    AND GVL_IO_WRITE_RUNTIME_BUFFER.B_Gas_Fire_Siren_Enable
    AND GVL_IO_WRITE_RUNTIME_BUFFER.B_Fire_Siren_Authority;

GVL_IO.DO_Security_Siren :=
    L_Audible_Siren_Allowed
    AND (
        GVL_ALARM.G_Security_Siren
        OR (GVL_ALARM.G_Global_Siren AND GVL_ALARM.G_Security_Alarm)
    );

GVL_IO.DO_Gas_Valve_Close := GVL_COMMAND_SHADOW.G_Gas_Valve_Close;

fbTrace(
    iLayer := TRACE_IO,
    iSource := SRC_IO,
    iReason := REASON_DOMAIN_PROJECTION,
    iValueBool := TRUE,
    iValueReal := 0.0,
    iText := 'IO write projection executed'
);

// >>> BULK_SYNC_ANCHOR: PRG_IO_Write_Phase_04_Alarm_Trace <<<
END_PROGRAM

(* ---- PRG_Lighting.st ---- *)
PROGRAM PRG_Lighting
// ==============================================================================
// LIGHTING — deterministic lighting/blinds/socket phase map.
// ==============================================================================
// Execution order is preserved from the former monolithic PRG_Lighting body.
// No gating, shedding or behavior changes are applied here.
// ==============================================================================

PRG_Lighting_Phase_01_Context();
PRG_Lighting_Phase_02_Managers();
PRG_Lighting_Phase_03_Priority_Restrictions();
PRG_Lighting_Phase_04_Output_Publication();

// >>> BULK_SYNC_ANCHOR: PRG_Lighting <<<
END_PROGRAM

(* ---- PRG_Lighting_Phase_01_Context.st ---- *)
PROGRAM PRG_Lighting_Phase_01_Context
VAR
    L_i : INT;
    L_Evac_Blink_Phase : UDINT;
END_VAR

GVL_LIGHTING_RUNTIME_BUFFER.B_Fire_Alarm_Active :=
    GVL_HEALTH_BRIDGE.G_Smoke_Detected
    OR GVL_STATE.G_Safety_Smoke_Latched;

GVL_LIGHTING_RUNTIME_BUFFER.B_Flood_Alarm_Active :=
    GVL_HEALTH_BRIDGE.G_Leak_Detected
    OR GVL_STATE.G_Safety_Leak_Latched;

GVL_LIGHTING_RUNTIME_BUFFER.B_Security_Armed := GVL_ALARM.G_Security_Armed;
GVL_LIGHTING_RUNTIME_BUFFER.B_Security_Alarm := GVL_ALARM.G_Security_Alarm;

L_Evac_Blink_Phase := (GVL_STATUS.G_System_Time_MS / 500) MOD 2;
GVL_LIGHTING_RUNTIME_BUFFER.B_Evac_Blink_On := (L_Evac_Blink_Phase = 0);

GVL_LIGHTING_RUNTIME_BUFFER.B_Distributed_Execute_Allowed :=
    GVL_Distributed_Execution_Gates.G_Can_Execute;

GVL_LIGHTING_RUNTIME_BUFFER.B_Distributed_Projection_Allowed :=
    GVL_Distributed_Execution_Gates.G_Can_Own_Projection;

GVL_LIGHTING_RUNTIME_BUFFER.B_Emergency_Lighting_Override :=
    GVL_STATE.G_Evacuation_Lighting_Active
    OR GVL_LIGHTING_RUNTIME_BUFFER.B_Fire_Alarm_Active;

FOR L_i := 1 TO GVL_CONSTANTS.C_MAX_LIGHT_ZONES DO
    IF GVL_INTENT_SYSTEM.I_Lighting_Overrides_Block OR GVL_SYSTEM_COORDINATION.G_Block_Lighting_Override THEN
        GVL_LIGHTING_RUNTIME_BUFFER.B_Manual_Light_Override[L_i] := 0;
    ELSE
        GVL_LIGHTING_RUNTIME_BUFFER.B_Manual_Light_Override[L_i] := GVL_INTENT_USER.I_Lighting_Override_32[L_i];
    END_IF;

    GVL_LIGHTING_RUNTIME_BUFFER.B_Sim_Lights[L_i] := GVL_STATE.G_Sim_Lights[L_i];
    GVL_LIGHTING_RUNTIME_BUFFER.B_Physical_Switches[L_i] := GVL_STATE.G_Physical_Switches[L_i];
    GVL_LIGHTING_RUNTIME_BUFFER.B_Motion_Sensors[L_i] := GVL_STATE.G_Motion_Sensors[L_i];

    IF GVL_INTENT_SYSTEM.I_Blinds_Overrides_Block THEN
        GVL_LIGHTING_RUNTIME_BUFFER.B_Manual_Blinds_Override[L_i] := 0;
    ELSE
        GVL_LIGHTING_RUNTIME_BUFFER.B_Manual_Blinds_Override[L_i] := GVL_INTENT_USER.I_Blinds_Override_32[L_i];
    END_IF;
END_FOR;

FOR L_i := 1 TO GVL_CONSTANTS.C_MAX_BLINDS DO
    GVL_LIGHTING_RUNTIME_BUFFER.B_Blinds_Override[L_i] :=
        GVL_LIGHTING_RUNTIME_BUFFER.B_Manual_Blinds_Override[L_i];
END_FOR;

FOR L_i := 1 TO GVL_CONSTANTS.C_MAX_SOCKETS DO
    IF GVL_INTENT_SYSTEM.I_Socket_Overrides_Block OR GVL_SYSTEM_COORDINATION.G_Block_Sockets_Override THEN
        GVL_LIGHTING_RUNTIME_BUFFER.B_Manual_Socket_Override[L_i] := FALSE;
    ELSE
        GVL_LIGHTING_RUNTIME_BUFFER.B_Manual_Socket_Override[L_i] := GVL_INTENT_USER.I_Socket_Override_32[L_i];
    END_IF;

    GVL_LIGHTING_RUNTIME_BUFFER.B_Socket_Override[L_i] :=
        GVL_LIGHTING_RUNTIME_BUFFER.B_Manual_Socket_Override[L_i];
END_FOR;

// >>> BULK_SYNC_ANCHOR: PRG_Lighting_Phase_01_Context <<<
END_PROGRAM

(* ---- PRG_Lighting_Phase_02_Managers.st ---- *)
PROGRAM PRG_Lighting_Phase_02_Managers
VAR
    fbLightingManager : FB_Lighting_Blinds_Manager;
    fbSocketManager : FB_Socket_Manager;
    fbOutdoorLightingManager : FB_Outdoor_Lighting_Manager;
    L_Effective_Rule_Actions : ARRAY[1..GVL_CONSTANTS.C_MAX_RULES] OF ST_Rule_Action;
    L_i : INT;
END_VAR

IF GVL_LIGHTING_RUNTIME_BUFFER.B_Distributed_Execute_Allowed THEN

    // Copy user/system rule actions into a cycle-local surface. Outdoor lighting
    // adds actions here so global GVL_STATE.G_Rule_Actions is not overwritten.
    FOR L_i := 1 TO GVL_CONSTANTS.C_MAX_RULES DO
        L_Effective_Rule_Actions[L_i] := GVL_STATE.G_Rule_Actions[L_i];
    END_FOR;

    fbOutdoorLightingManager(
        VI_IsActivePLC := GVL_STATUS.G_Is_Active_PLC,
        VI_Current_Scenario := GVL_STATUS.G_Current_Scenario,
        VI_Security_Armed := GVL_ALARM.G_Security_Armed,
        VI_Is_Night := GVL_STATUS.G_Is_Night,
        VI_Time_Of_Day_MS := GVL_TIME_SERVICE.G_Time_Of_Day_MS,
        VIO_Rule_Actions := L_Effective_Rule_Actions,
        VI_Motion_Sensors := GVL_LIGHTING_RUNTIME_BUFFER.B_Motion_Sensors
    );

    fbLightingManager(
        VI_System_Time_MS := GVL_STATUS.G_System_Time_MS,
        VI_IsActivePLC := GVL_STATUS.G_Is_Active_PLC,
        VI_Current_Scenario := GVL_STATUS.G_Current_Scenario,
        VI_Away_Level := GVL_POLICY.G_Away_Level,
        VI_Simulation_Active := GVL_STATUS.G_Sim_Active OR GVL_POLICY.G_Away_Simulation_Active,
        VI_Is_Night := GVL_STATUS.G_Is_Night,
        VI_System_Mode := GVL_STATE.G_System_Mode,
        VI_Manual_Light_Override := GVL_LIGHTING_RUNTIME_BUFFER.B_Manual_Light_Override,
        VI_Manual_Blinds_Override := GVL_LIGHTING_RUNTIME_BUFFER.B_Blinds_Override,
        VI_Simulation_Lights := GVL_LIGHTING_RUNTIME_BUFFER.B_Sim_Lights,
        VI_Physical_Switches := GVL_LIGHTING_RUNTIME_BUFFER.B_Physical_Switches,
        VI_Motion_Sensors := GVL_LIGHTING_RUNTIME_BUFFER.B_Motion_Sensors,
        VI_Rule_Actions := L_Effective_Rule_Actions,
        VI_IO_Modules_Online := GVL_STATUS.G_IO_Modules_Online,
        VI_Wet_Zone_Map := GVL_CONFIG.G_Wet_Zone_Map,
        VI_Scenario_Configs := GVL_CONFIG.G_HMI_Scenario_Configs,
        VO_Lighting_Levels => GVL_STATE.G_Lighting_Levels,
        VO_Blinds_Positions => GVL_STATE.G_Blinds_Positions,
        VO_Wet_Zone_Light_Active => GVL_LIGHTING_RUNTIME_BUFFER.B_Wet_Zone_Light_Active
    );

    fbSocketManager(
        VI_System_Time_MS := GVL_STATUS.G_System_Time_MS,
        VI_IsActivePLC := GVL_STATUS.G_Is_Active_PLC,
        VI_Scenario := GVL_STATUS.G_Current_Scenario,
        VI_Manual_Override := GVL_LIGHTING_RUNTIME_BUFFER.B_Socket_Override,
        VI_Physical_Switches := GVL_STATE.G_Socket_Switches,
        VI_Rule_Actions := L_Effective_Rule_Actions,
        VI_Fire_Alarm := GVL_LIGHTING_RUNTIME_BUFFER.B_Fire_Alarm_Active,
        VI_Flood_Alarm := GVL_LIGHTING_RUNTIME_BUFFER.B_Flood_Alarm_Active,
        VI_Security_Armed := GVL_ALARM.G_Security_Armed,
        VI_IO_Modules_Online := GVL_STATUS.G_IO_Modules_Online,
        VO_Socket_States => GVL_STATE.G_Socket_States
    );

END_IF;

// >>> BULK_SYNC_ANCHOR: PRG_Lighting_Phase_02_Managers <<<
END_PROGRAM

(* ---- PRG_Lighting_Phase_03_Priority_Restrictions.st ---- *)
PROGRAM PRG_Lighting_Phase_03_Priority_Restrictions
VAR
    L_i : INT;
END_VAR

// Priority overrides after normal manager calculation:
// Evacuation > Fire > Security Alarm > Security Armed > Normal
IF GVL_STATE.G_Evacuation_Lighting_Active THEN
    FOR L_i := 1 TO GVL_CONSTANTS.C_MAX_LIGHT_ZONES DO
        CASE GVL_STATE.G_Evac_Guidance[L_i] OF
            -1:
                GVL_STATE.G_Lighting_Levels[L_i] := 0;
            1:
                GVL_STATE.G_Lighting_Levels[L_i] := 100;
        ELSE
            IF GVL_LIGHTING_RUNTIME_BUFFER.B_Evac_Blink_On THEN
                GVL_STATE.G_Lighting_Levels[L_i] := 100;
            ELSE
                GVL_STATE.G_Lighting_Levels[L_i] := 0;
            END_IF;
        END_CASE;
    END_FOR;
ELSIF GVL_LIGHTING_RUNTIME_BUFFER.B_Fire_Alarm_Active THEN
    FOR L_i := 1 TO GVL_CONSTANTS.C_MAX_LIGHT_ZONES DO
        GVL_STATE.G_Lighting_Levels[L_i] := 100;
    END_FOR;
    FOR L_i := 1 TO GVL_CONSTANTS.C_MAX_BLINDS DO
        GVL_STATE.G_Blinds_Positions[L_i] := 100;
    END_FOR;
ELSIF GVL_LIGHTING_RUNTIME_BUFFER.B_Security_Alarm THEN
    FOR L_i := 1 TO GVL_CONSTANTS.C_MAX_LIGHT_ZONES DO
        GVL_STATE.G_Lighting_Levels[L_i] := 100;
    END_FOR;
ELSIF GVL_LIGHTING_RUNTIME_BUFFER.B_Security_Armed THEN
    FOR L_i := 1 TO GVL_CONSTANTS.C_MAX_LIGHT_ZONES DO
        GVL_STATE.G_Lighting_Levels[L_i] := 0;
    END_FOR;
END_IF;

// Distributed projection restriction.
IF NOT GVL_LIGHTING_RUNTIME_BUFFER.B_Distributed_Projection_Allowed
   AND NOT GVL_LIGHTING_RUNTIME_BUFFER.B_Emergency_Lighting_Override THEN

    FOR L_i := 1 TO GVL_CONSTANTS.C_MAX_LIGHT_ZONES DO
        GVL_STATE.G_Lighting_Levels[L_i] := 0;
    END_FOR;

    FOR L_i := 1 TO GVL_CONSTANTS.C_MAX_BLINDS DO
        GVL_STATE.G_Blinds_Positions[L_i] := 100;
    END_FOR;

    FOR L_i := 1 TO GVL_CONSTANTS.C_MAX_SOCKETS DO
        GVL_STATE.G_Socket_States[L_i] := FALSE;
    END_FOR;

END_IF;

// >>> BULK_SYNC_ANCHOR: PRG_Lighting_Phase_03_Priority_Restrictions <<<
END_PROGRAM

(* ---- PRG_Lighting_Phase_04_Output_Publication.st ---- *)
PROGRAM PRG_Lighting_Phase_04_Output_Publication
VAR
    L_i : INT;
    L_Wet_Zone_Any_Active : BOOL;
END_VAR

// Publish wet-zone activity from the final lighting state seen by IO_Write.
L_Wet_Zone_Any_Active := FALSE;
FOR L_i := 1 TO GVL_CONSTANTS.C_MAX_LIGHT_ZONES DO
    IF GVL_CONFIG.G_Wet_Zone_Map[L_i] AND (GVL_STATE.G_Lighting_Levels[L_i] > 10) THEN
        L_Wet_Zone_Any_Active := TRUE;
    END_IF;
END_FOR;
GVL_STATUS.G_Wet_Zone_Light_Active := L_Wet_Zone_Any_Active;

// Domain output projection.
FOR L_i := 1 TO GVL_CONSTANTS.C_MAX_LIGHT_ZONES DO
    GVL_LIGHTING_OUTPUT.AO_Lighting_Levels[L_i] := BYTE_TO_UINT(GVL_STATE.G_Lighting_Levels[L_i]) * 10;
END_FOR;

FOR L_i := 1 TO GVL_CONSTANTS.C_MAX_BLINDS DO
    GVL_LIGHTING_OUTPUT.AO_Blinds_Positions[L_i] := BYTE_TO_UINT(GVL_STATE.G_Blinds_Positions[L_i]) * 10;
END_FOR;

FOR L_i := 1 TO GVL_CONSTANTS.C_MAX_SOCKETS DO
    GVL_LIGHTING_OUTPUT.DO_Sockets[L_i] := GVL_STATE.G_Socket_States[L_i];
END_FOR;

// >>> BULK_SYNC_ANCHOR: PRG_Lighting_Phase_04_Output_Publication <<<
END_PROGRAM

(* ---- PRG_Main_Feedback_Mark_04.st ---- *)
PROGRAM PRG_Main_Feedback_Mark_04
GVL_MAIN_PHASE_FEEDBACK.G_Phase_04_Transport_Distributed_Executed := TRUE;
GVL_MAIN_PHASE_FEEDBACK.G_Phase_04_Transport_Distributed_Valid := TRUE;
GVL_MAIN_PHASE_FEEDBACK.G_Phase_04_Transport_Distributed_Status_Text := 'Transport/distributed phase executed';
GVL_MAIN_PHASE_FEEDBACK.G_Last_Update_MS := GVL_TIME_SERVICE.G_Now_MS;
END_PROGRAM

(* ---- PRG_Main_Feedback_Mark_05.st ---- *)
PROGRAM PRG_Main_Feedback_Mark_05
GVL_MAIN_PHASE_FEEDBACK.G_Phase_05_Domain_Output_Executed := TRUE;
GVL_MAIN_PHASE_FEEDBACK.G_Phase_05_Domain_Output_Valid := TRUE;
GVL_MAIN_PHASE_FEEDBACK.G_Phase_05_Domain_Output_Status_Text := 'Domain/output phase executed';
GVL_MAIN_PHASE_FEEDBACK.G_Last_Update_MS := GVL_TIME_SERVICE.G_Now_MS;
END_PROGRAM

(* ---- PRG_Main_Feedback_Mark_06.st ---- *)
PROGRAM PRG_Main_Feedback_Mark_06
GVL_MAIN_PHASE_FEEDBACK.G_Phase_06_PostOutput_Authority_Executed := TRUE;
GVL_MAIN_PHASE_FEEDBACK.G_Phase_06_PostOutput_Authority_Valid := TRUE;
GVL_MAIN_PHASE_FEEDBACK.G_Phase_06_PostOutput_Authority_Status_Text := 'Post-output authority phase executed';
GVL_MAIN_PHASE_FEEDBACK.G_Last_Update_MS := GVL_TIME_SERVICE.G_Now_MS;
END_PROGRAM

(* ---- PRG_Main_Feedback_Mark_07.st ---- *)
PROGRAM PRG_Main_Feedback_Mark_07
GVL_MAIN_PHASE_FEEDBACK.G_Phase_07_Semantic_Governance_Executed := TRUE;
GVL_MAIN_PHASE_FEEDBACK.G_Phase_07_Semantic_Governance_Valid := TRUE;
GVL_MAIN_PHASE_FEEDBACK.G_Phase_07_Semantic_Governance_Status_Text := 'Semantic/governance phase executed';
GVL_MAIN_PHASE_FEEDBACK.G_Last_Update_MS := GVL_TIME_SERVICE.G_Now_MS;
END_PROGRAM

(* ---- PRG_Main_Phase_01_Bootstrap.st ---- *)
PROGRAM PRG_Main_Phase_01_Bootstrap
// MAIN PHASE 01/02 — time, configuration and canonical runtime baseline.
// Critical: yes. Called every PLC scan.

GVL_MAIN_PHASE_FEEDBACK.G_Current_Phase := 1;

// Reset observational phase feedback at the beginning of every PLC scan.
GVL_MAIN_PHASE_FEEDBACK.G_Phase_01_Bootstrap_Executed := FALSE;
GVL_MAIN_PHASE_FEEDBACK.G_Phase_01_Bootstrap_Valid := FALSE;
GVL_MAIN_PHASE_FEEDBACK.G_Phase_01_Bootstrap_Status_Text := '';

GVL_MAIN_PHASE_FEEDBACK.G_Phase_02_Redundancy_Executed := FALSE;
GVL_MAIN_PHASE_FEEDBACK.G_Phase_02_Redundancy_Valid := FALSE;
GVL_MAIN_PHASE_FEEDBACK.G_Phase_02_Redundancy_Status_Text := '';

GVL_MAIN_PHASE_FEEDBACK.G_Phase_03_Input_Safety_Command_Executed := FALSE;
GVL_MAIN_PHASE_FEEDBACK.G_Phase_03_Input_Safety_Command_Valid := FALSE;
GVL_MAIN_PHASE_FEEDBACK.G_Phase_03_Input_Safety_Command_Status_Text := '';

GVL_MAIN_PHASE_FEEDBACK.G_Phase_04_Transport_Distributed_Executed := FALSE;
GVL_MAIN_PHASE_FEEDBACK.G_Phase_04_Transport_Distributed_Valid := FALSE;
GVL_MAIN_PHASE_FEEDBACK.G_Phase_04_Transport_Distributed_Status_Text := '';

GVL_MAIN_PHASE_FEEDBACK.G_Phase_05_Domain_Output_Executed := FALSE;
GVL_MAIN_PHASE_FEEDBACK.G_Phase_05_Domain_Output_Valid := FALSE;
GVL_MAIN_PHASE_FEEDBACK.G_Phase_05_Domain_Output_Status_Text := '';

GVL_MAIN_PHASE_FEEDBACK.G_Phase_06_PostOutput_Authority_Executed := FALSE;
GVL_MAIN_PHASE_FEEDBACK.G_Phase_06_PostOutput_Authority_Valid := FALSE;
GVL_MAIN_PHASE_FEEDBACK.G_Phase_06_PostOutput_Authority_Status_Text := '';

GVL_MAIN_PHASE_FEEDBACK.G_Phase_07_Semantic_Governance_Executed := FALSE;
GVL_MAIN_PHASE_FEEDBACK.G_Phase_07_Semantic_Governance_Valid := FALSE;
GVL_MAIN_PHASE_FEEDBACK.G_Phase_07_Semantic_Governance_Status_Text := '';

GVL_MAIN_PHASE_FEEDBACK.G_Phase_07_Full_Semantic_Requested := FALSE;
GVL_MAIN_PHASE_FEEDBACK.G_Phase_07_Full_Semantic_Executed := FALSE;
GVL_MAIN_PHASE_FEEDBACK.G_Phase_07_Full_Semantic_Skipped_By_Design := FALSE;
GVL_MAIN_PHASE_FEEDBACK.G_Phase_07_Extended_Observability_Requested := FALSE;
GVL_MAIN_PHASE_FEEDBACK.G_Phase_07_Extended_Observability_Executed := FALSE;
GVL_MAIN_PHASE_FEEDBACK.G_Phase_07_Extended_Observability_Skipped_By_Design := FALSE;
GVL_MAIN_PHASE_FEEDBACK.G_Phase_07_Analytics_Requested := FALSE;
GVL_MAIN_PHASE_FEEDBACK.G_Phase_07_Analytics_Executed := FALSE;
GVL_MAIN_PHASE_FEEDBACK.G_Phase_07_Analytics_Skipped_By_Design := FALSE;

GVL_MAIN_PHASE_FEEDBACK.G_Phase_08_Diagnostics_HMI_Executed := FALSE;
GVL_MAIN_PHASE_FEEDBACK.G_Phase_08_Diagnostics_HMI_Valid := FALSE;
GVL_MAIN_PHASE_FEEDBACK.G_Phase_08_Diagnostics_HMI_Status_Text := '';

GVL_MAIN_PHASE_FEEDBACK.G_Phase_08_Extended_Diagnostics_Requested := FALSE;
GVL_MAIN_PHASE_FEEDBACK.G_Phase_08_Extended_Diagnostics_Executed := FALSE;
GVL_MAIN_PHASE_FEEDBACK.G_Phase_08_Extended_Diagnostics_Skipped_By_Design := FALSE;
GVL_MAIN_PHASE_FEEDBACK.G_Phase_08_Extended_Observability_Requested := FALSE;
GVL_MAIN_PHASE_FEEDBACK.G_Phase_08_Extended_Observability_Executed := FALSE;
GVL_MAIN_PHASE_FEEDBACK.G_Phase_08_Extended_Observability_Skipped_By_Design := FALSE;
GVL_MAIN_PHASE_FEEDBACK.G_Phase_08_Simulation_Requested := FALSE;
GVL_MAIN_PHASE_FEEDBACK.G_Phase_08_Simulation_Executed := FALSE;
GVL_MAIN_PHASE_FEEDBACK.G_Phase_08_Simulation_Skipped_By_Design := FALSE;

GVL_MAIN_PHASE_FEEDBACK.G_Critical_Path_Executed := FALSE;
GVL_MAIN_PHASE_FEEDBACK.G_Critical_Path_Valid := FALSE;
GVL_MAIN_PHASE_FEEDBACK.G_Observability_Path_Executed := FALSE;
GVL_MAIN_PHASE_FEEDBACK.G_Observability_Path_Valid := FALSE;
GVL_MAIN_PHASE_FEEDBACK.G_Any_Phase_Invalid := FALSE;
GVL_MAIN_PHASE_FEEDBACK.G_Any_Phase_Skipped_By_Design := FALSE;
GVL_MAIN_PHASE_FEEDBACK.G_Status_Code := 0;
GVL_MAIN_PHASE_FEEDBACK.G_Status_Text := 'MAIN phase feedback reset';

PRG_Time_Service();
PRG_Time_Monotonic_Governor();

GVL_MAIN_PHASE_FEEDBACK.G_Cycle_Start_MS := GVL_TIME_SERVICE.G_Now_MS;

PRG_System_Init();
PRG_Config_Manager();
PRG_Config_Validation();
PRG_Config_Versioning();
PRG_System_Runtime_Base();

PRG_Temporal_Domain();
PRG_Runtime_Core_Domain();
PRG_Safety_Domain();
PRG_Recovery_Domain();
PRG_Distributed_Domain();
PRG_Verification_Domain();
PRG_Semantic_Commit_Governor();

GVL_MAIN_PHASE_FEEDBACK.G_Phase_01_Bootstrap_Executed := TRUE;
GVL_MAIN_PHASE_FEEDBACK.G_Phase_01_Bootstrap_Valid := TRUE;
GVL_MAIN_PHASE_FEEDBACK.G_Phase_01_Bootstrap_Status_Text := 'Bootstrap/runtime baseline executed';
GVL_MAIN_PHASE_FEEDBACK.G_Last_Update_MS := GVL_TIME_SERVICE.G_Now_MS;

// >>> BULK_SYNC_ANCHOR: PRG_Main_Phase_01_Bootstrap <<<
END_PROGRAM

(* ---- PRG_Main_Phase_02_Redundancy.st ---- *)
PROGRAM PRG_Main_Phase_02_Redundancy
// MAIN PHASE 03 — redundancy, heartbeat and active/standby arbitration.
// Critical: yes. Called every PLC scan.
VAR
    fbSystemRedundancyOrchestrator : FB_System_Redundancy_Orchestrator;
    fbSystemDiagnostics : FB_System_Diagnostics;
    fbStateReplication : FB_State_Replication;
    fbRedundancyManager : FB_Redundancy_Manager;
    fbPLCHeartbeat : FB_PLC_Heartbeat;

    L_Main_Local_State : ST_System_State_Snapshot;
    L_Main_Remote_State : ST_System_State_Snapshot;
    L_Main_Synced_State : ST_System_State_Snapshot;
    L_Main_State_Updated : BOOL;
    L_Main_PLC_Active : BOOL;
    L_Main_RTT_MS : UDINT;
    L_Main_Loss_Count : UDINT;
    L_Main_Max_RTT : UDINT;
END_VAR

GVL_MAIN_PHASE_FEEDBACK.G_Current_Phase := 2;

fbPLCHeartbeat(
    VI_Local_ID := GVL_STATUS.G_PLC_ID,
    VI_System_Time := GVL_STATUS.G_System_Time_MS,
    VI_Remote_Pulse := GVL_IO.DI_Partner_Pulse,
    VI_Remote_Is_Active := GVL_IO.DI_Partner_Active,
    VI_Gateway_Ping_OK := GVL_GATEWAY.G_Gateway_Ping_OK,
    VO_Is_Active => L_Main_PLC_Active,
    VO_RTT_MS => L_Main_RTT_MS,
    VO_Loss_Count => L_Main_Loss_Count,
    VO_Max_RTT => L_Main_Max_RTT
);

fbStateReplication(
    VI_Local_Role := SEL(GVL_STATUS.G_Is_Active_PLC, E_PLC_ROLE.ROLE_STANDBY, E_PLC_ROLE.ROLE_ACTIVE),
    VI_Sync_Req := FALSE,
    VI_Local_State := L_Main_Local_State,
    VI_Remote_State := L_Main_Remote_State,
    VI_System_Time_MS := GVL_STATUS.G_System_Time_MS,
    VO_State_Updated => L_Main_State_Updated,
    VO_Synced_State => L_Main_Synced_State
);

fbRedundancyManager(
    VI_System_Time_MS := GVL_STATUS.G_System_Time_MS,
    VI_Local_PLC_ID := GVL_STATUS.G_PLC_ID,
    VI_Remote_Pulse := GVL_IO.DI_Partner_Pulse,
    VI_Remote_Is_Active := GVL_IO.DI_Partner_Active,
    VI_Gateway_Ping_OK := GVL_GATEWAY.G_Gateway_Ping_OK,
    VI_Local_State := L_Main_Local_State,
    VI_Remote_State := L_Main_Remote_State
);

fbSystemDiagnostics();

fbSystemRedundancyOrchestrator(
    VIO_Local_State := L_Main_Local_State,
    VIO_Remote_State := L_Main_Remote_State
);

PRG_Peer_Heartbeat_Ingestion();
PRG_PLC_Arbitration();
PRG_PLC_Fencing_Governor();

GVL_MAIN_PHASE_FEEDBACK.G_Phase_02_Redundancy_Executed := TRUE;
GVL_MAIN_PHASE_FEEDBACK.G_Phase_02_Redundancy_Valid := TRUE;
GVL_MAIN_PHASE_FEEDBACK.G_Phase_02_Redundancy_Status_Text := 'Redundancy/heartbeat phase executed';
GVL_MAIN_PHASE_FEEDBACK.G_Last_Update_MS := GVL_TIME_SERVICE.G_Now_MS;

// >>> BULK_SYNC_ANCHOR: PRG_Main_Phase_02_Redundancy <<<
END_PROGRAM

(* ---- PRG_Main_Phase_03_Input_Safety_Command.st ---- *)
PROGRAM PRG_Main_Phase_03_Input_Safety_Command
VAR
END_VAR

GVL_MAIN_PHASE_FEEDBACK.G_Current_Phase := 3;

PRG_IO_Read();
PRG_Input_Quality_Read();
PRG_Input_Processing();

PRG_Mode_Manager();
PRG_Presence_Manager();
PRG_Safety_Selector();
PRG_Safety();
PRG_Safety_Operator();
PRG_Safety_Shutdown();
PRG_Safety_Recovery();
PRG_System_Intent();
PRG_Security();
PRG_System_Access_Maintenance();
PRG_User_Adapt_Control();
PRG_Behavior_Adapt_Profile();

PRG_Scenario_Engine();
PRG_System_Scenario_Rules();
PRG_System_Evacuation();
PRG_Policy();
PRG_Heating_Policy_Manager();
PRG_Heating_Policy_Observer();
PRG_System_Coordinator();
PRG_Command_Arbitration();

GVL_MAIN_PHASE_FEEDBACK.G_Phase_03_Input_Safety_Command_Executed := TRUE;
GVL_MAIN_PHASE_FEEDBACK.G_Phase_03_Input_Safety_Command_Valid := TRUE;
GVL_MAIN_PHASE_FEEDBACK.G_Phase_03_Input_Safety_Command_Status_Text := 'Input/safety/command phase executed';
GVL_MAIN_PHASE_FEEDBACK.G_Last_Update_MS := GVL_TIME_SERVICE.G_Now_MS;

// >>> BULK_SYNC_ANCHOR: PRG_Main_Phase_03_Input_Safety_Command <<<
END_PROGRAM

(* ---- PRG_Main_Phase_04_Transport_Distributed.st ---- *)
PROGRAM PRG_Main_Phase_04_Transport_Distributed
// MAIN PHASE 07/08 — fieldbus, transport, runtime barriers and distributed governance.
// Critical: mixed. Transport/barrier parts are runtime-critical; observability parts can be reviewed later for shedding.

GVL_MAIN_PHASE_FEEDBACK.G_Current_Phase := 4;

PRG_Modbus_Master();
PRG_Modbus_RTU_Bridge();
PRG_Modbus_RTU_Driver();
PRG_Modbus_RTU_SysCom_Backend();
PRG_Modbus_RTU_SysCom_Transport();
PRG_Modbus_Register_Scan();
PRG_OpenTherm_Command_Interface();
PRG_OpenTherm_Transport();
PRG_OpenTherm_Adapter_Status();
PRG_Transport_Freshness_Governor();

PRG_Runtime_Barrier();
PRG_Runtime_Snapshot_Governor();
PRG_Peer_Session_Publication();
PRG_HA_Session_Replication();
PRG_Distributed_Peer_Ingestion();
PRG_Distributed_Epoch_Governor();
PRG_Distributed_Snapshot_Publication();
PRG_Distributed_Snapshot_Ingestion();
PRG_Distributed_Snapshot_Governor();
PRG_Distributed_Runtime_Supervisor();
PRG_Distributed_Commit_Publication();
PRG_Distributed_Commit_Ingestion();
PRG_Distributed_Commit_Governor();
PRG_Distributed_Commit_Observability();
PRG_Semantic_Progress_Governor();
PRG_Convergence_Governor();
PRG_Recovery_Cleanup_Governor();
PRG_Observability_Governor();

GVL_MAIN_PHASE_FEEDBACK.G_Phase_04_Transport_Distributed_Executed := TRUE;
GVL_MAIN_PHASE_FEEDBACK.G_Phase_04_Transport_Distributed_Valid := TRUE;
GVL_MAIN_PHASE_FEEDBACK.G_Phase_04_Transport_Distributed_Status_Text := 'Transport/distributed phase executed';
GVL_MAIN_PHASE_FEEDBACK.G_Last_Update_MS := GVL_TIME_SERVICE.G_Now_MS;

// >>> BULK_SYNC_ANCHOR: PRG_Main_Phase_04_Transport_Distributed <<<
END_PROGRAM

(* ---- PRG_Main_Phase_05_Domain_Output.st ---- *)
PROGRAM PRG_Main_Phase_05_Domain_Output
// MAIN PHASE 09/10/11 — domain control, output validation and physical IO projection.
// Critical: yes. This is the physical actuation path and must run every PLC scan.

GVL_MAIN_PHASE_FEEDBACK.G_Current_Phase := 5;

PRG_Heating();
PRG_Heating_Supervisory_Publication();
PRG_Ventilation();
PRG_Water_Supervisory_Publication();
PRG_Water_Output_Projection();
PRG_Water();
PRG_Access();
PRG_Lighting();

// Observational execution-demand matrix.
// Reads the already calculated domain outputs/statuses from this scan.
// Does not gate execution yet.
PRG_Domain_Execution_Policy();

PRG_Output_Freshness_Governor();
PRG_Physical_Snapshot_Governor();
PRG_Sensor_Consensus_Governor();
PRG_Telemetry_Causality_Governor();
PRG_Physical_Authority_Epoch_Governor();
PRG_Authority_Lineage_Governor();
PRG_Authority_Revocation_Governor();
PRG_Authority_Restoration_Governor();

PRG_PreOutput_Safety_Barrier();
PRG_IO_Write();

GVL_MAIN_PHASE_FEEDBACK.G_Phase_05_Domain_Output_Executed := TRUE;
GVL_MAIN_PHASE_FEEDBACK.G_Phase_05_Domain_Output_Valid := TRUE;
GVL_MAIN_PHASE_FEEDBACK.G_Phase_05_Domain_Output_Status_Text := 'Domain/output phase executed';
GVL_MAIN_PHASE_FEEDBACK.G_Last_Update_MS := GVL_TIME_SERVICE.G_Now_MS;

// >>> BULK_SYNC_ANCHOR: PRG_Main_Phase_05_Domain_Output <<<
END_PROGRAM

(* ---- PRG_Main_Phase_06_PostOutput_Authority.st ---- *)
PROGRAM PRG_Main_Phase_06_PostOutput_Authority
// MAIN PHASE 12A — post-output authority, physical transaction and causality guards.
// Critical: high. Runs after IO projection to validate authority/physical consistency.

PRG_Actuation_Authority_Governor();
PRG_Physical_Transaction_Governor();
PRG_Temporal_Stability_Governor();
PRG_Environmental_Authority_Governor();
PRG_Runtime_Resource_Authority_Governor();
PRG_Semantic_Continuity_Authority_Governor();
PRG_Observability_Truth_Governor();
PRG_Historical_Truth_Governor();
PRG_Global_Authority_Sync_Governor();
PRG_Control_Temporal_Coherence_Governor();
PRG_Actuator_Semantic_Verification_Governor();
PRG_Energy_Causality_Governor();
PRG_Runtime_Sustainability_Governor();

// >>> BULK_SYNC_ANCHOR: PRG_Main_Phase_06_PostOutput_Authority <<<
END_PROGRAM

(* ---- PRG_Main_Phase_07_Semantic_Governance.st ---- *)
PROGRAM PRG_Main_Phase_07_Semantic_Governance
// MAIN PHASE 12B — semantic, forensic, recovery, energy and governance integrity.
// Critical: mixed. Safety/authority/physical reality checks run every scan.
// Non-critical semantic, forensic and analytics fabrics are shed in reduced modes.
VAR
    L_Run_Full_Semantic : BOOL;
    L_Run_Extended_Observability : BOOL;
    L_Run_Analytics : BOOL;
END_VAR

GVL_MAIN_PHASE_FEEDBACK.G_Current_Phase := 7;

L_Run_Full_Semantic :=
    GVL_FABRIC_LIFECYCLE_REGISTRY.Runtime_Adaptive_Mode = FULL_SEMANTIC_MODE;

L_Run_Extended_Observability :=
    (GVL_FABRIC_LIFECYCLE_REGISTRY.Runtime_Adaptive_Mode = FULL_SEMANTIC_MODE)
    AND NOT GVL_FABRIC_LIFECYCLE_REGISTRY.Extended_Observability_Shedding_Recommended;

L_Run_Analytics :=
    (GVL_FABRIC_LIFECYCLE_REGISTRY.Runtime_Adaptive_Mode = FULL_SEMANTIC_MODE)
    AND NOT GVL_FABRIC_LIFECYCLE_REGISTRY.NonEssential_Analytics_Shedding_Recommended;

// Critical authority and physical-reality guards: never shed here.
PRG_Authority_Provenance_Governor();
PRG_Provenance_Continuity_Governor();
PRG_Trust_Epoch_Monotonicity_Governor();
PRG_Governance_Publication_Binding_Governor();
PRG_Physical_SafeState_Lattice_Governor();
PRG_CrossDomain_FailSafe_Closure_Governor();
PRG_Deterministic_Recovery_Path_Governor();
PRG_Recovery_Ordering_Integrity_Governor();
PRG_Recovery_Reactivation_Control_Governor();
PRG_Authority_Resurrection_Boundary_Governor();
PRG_Energy_Isolation_Causality_Governor();
PRG_Residual_Energy_State_Governor();
PRG_Power_Domain_Segmentation_Governor();
PRG_Energy_Resurrection_Boundary_Governor();
PRG_Physical_Deadlock_Resolution_Governor();
PRG_Execution_Progress_Causality_Governor();
PRG_Resource_Starvation_Boundary_Governor();
PRG_Distributed_Forward_Progress_Governor();
PRG_Safety_Observability_Truth_Governor();
PRG_Physical_Safety_Projection_Governor();
PRG_Distributed_Safety_Reality_Consensus_Governor();
PRG_Temporal_Causality_Closure_Governor();
PRG_Distributed_Epoch_Linearity_Governor();
PRG_Historical_Ordering_Integrity_Governor();
PRG_Causality_Reversal_Prevention_Governor();
PRG_Runtime_Transition_Validator();
PRG_Physical_Reality_Validation_Governor();
PRG_Survivability_Intelligence_Governor();
PRG_Runtime_Budget_Governor();
PRG_Controlled_Capability_Shedding_Governor();
PRG_Semantic_Execution_Control_Governor();
PRG_Industrial_Maintainability_Governor();
PRG_Observability_Authority_Governor();

// Full semantic fabrics: shed outside FULL_SEMANTIC_MODE.
IF L_Run_Full_Semantic THEN
    PRG_Semantic_Preservation_Governor();
    PRG_Operator_Semantic_Alignment_Governor();
    PRG_Semantic_Federation_Governor();
    PRG_Compliance_Federation_Governor();
    PRG_Epistemic_Integrity_Governor();
    PRG_Meta_Governance_Governor();
    PRG_Semantic_Epoch_Invariance_Governor();
    PRG_Governance_Observer_Consensus_Governor();
    PRG_Governance_Feedback_Integrity_Governor();
    PRG_Governance_Validator_Integrity_Governor();
    PRG_Governance_Liveness_Integrity_Governor();
    PRG_Runtime_Assumption_Integrity_Governor();
END_IF;

// Extended observability and forensic fabrics: shed when observability budget is constrained.
IF L_Run_Extended_Observability THEN
    PRG_Forensic_Evidence_Governor();
    PRG_Unsafe_Transition_Forensics_Governor();
    PRG_Passive_Runtime_Verification_Governor();
    PRG_Semantic_Drift_Observability_Governor();
    PRG_Proof_Continuity_Audit_Governor();
    PRG_Causal_Narrative_Engine();
END_IF;

// Non-essential analytics/intelligence fabrics: shed when analytics budget is constrained.
IF L_Run_Analytics THEN
    PRG_Execution_Projection_Integrity_Governor();
    PRG_Operational_Intelligence_Governor();
    PRG_Runtime_Compression_Governor();
END_IF;

GVL_MAIN_PHASE_FEEDBACK.G_Phase_07_Semantic_Governance_Executed := TRUE;
GVL_MAIN_PHASE_FEEDBACK.G_Phase_07_Semantic_Governance_Valid := TRUE;

IF L_Run_Full_Semantic AND L_Run_Extended_Observability AND L_Run_Analytics THEN
    GVL_MAIN_PHASE_FEEDBACK.G_Phase_07_Semantic_Governance_Status_Text := 'Semantic/governance phase executed';
ELSE
    GVL_MAIN_PHASE_FEEDBACK.G_Phase_07_Semantic_Governance_Status_Text := 'Semantic/governance phase executed with shedding';
END_IF;

GVL_MAIN_PHASE_FEEDBACK.G_Last_Update_MS := GVL_TIME_SERVICE.G_Now_MS;

// >>> BULK_SYNC_ANCHOR: PRG_Main_Phase_07_Semantic_Governance <<<
END_PROGRAM

(* ---- PRG_Main_Phase_08_Diagnostics_HMI.st ---- *)
PROGRAM PRG_Main_Phase_08_Diagnostics_HMI
// MAIN PHASE 13 — verification, explainability, diagnostics, history, simulation, HMI and debug.
// Critical: mixed. Command verification, health, alarm and debug summary remain active.
// History/trend/blackbox/simulation are shed when runtime budget asks for reduced work.
VAR
    L_Run_Extended_Diagnostics : BOOL;
    L_Run_Extended_Observability : BOOL;
    L_Run_Simulation : BOOL;
END_VAR

GVL_MAIN_PHASE_FEEDBACK.G_Current_Phase := 8;

L_Run_Extended_Diagnostics :=
    NOT GVL_FABRIC_LIFECYCLE_REGISTRY.Diagnostics_Degradation_Recommended;

L_Run_Extended_Observability :=
    (GVL_FABRIC_LIFECYCLE_REGISTRY.Runtime_Adaptive_Mode = FULL_SEMANTIC_MODE)
    AND NOT GVL_FABRIC_LIFECYCLE_REGISTRY.Extended_Observability_Shedding_Recommended;

L_Run_Simulation :=
    (GVL_FABRIC_LIFECYCLE_REGISTRY.Runtime_Adaptive_Mode = FULL_SEMANTIC_MODE)
    AND NOT GVL_FABRIC_LIFECYCLE_REGISTRY.Simulation_Suspension_Recommended;

GVL_MAIN_PHASE_FEEDBACK.G_Phase_08_Extended_Diagnostics_Requested := L_Run_Extended_Diagnostics;
GVL_MAIN_PHASE_FEEDBACK.G_Phase_08_Extended_Diagnostics_Executed := FALSE;
GVL_MAIN_PHASE_FEEDBACK.G_Phase_08_Extended_Diagnostics_Skipped_By_Design := NOT L_Run_Extended_Diagnostics;

GVL_MAIN_PHASE_FEEDBACK.G_Phase_08_Extended_Observability_Requested := L_Run_Extended_Observability;
GVL_MAIN_PHASE_FEEDBACK.G_Phase_08_Extended_Observability_Executed := FALSE;
GVL_MAIN_PHASE_FEEDBACK.G_Phase_08_Extended_Observability_Skipped_By_Design := NOT L_Run_Extended_Observability;

GVL_MAIN_PHASE_FEEDBACK.G_Phase_08_Simulation_Requested := L_Run_Simulation;
GVL_MAIN_PHASE_FEEDBACK.G_Phase_08_Simulation_Executed := FALSE;
GVL_MAIN_PHASE_FEEDBACK.G_Phase_08_Simulation_Skipped_By_Design := NOT L_Run_Simulation;

// Always-active verification, explainability, health, alarms, basic diagnostics and HMI/debug summary.
PRG_Command_Verifier();
PRG_Explainability();
PRG_System_Health();
PRG_System_Alarm_Gateway();
PRG_System_Diagnostics();
PRG_HMI_Dashboard();
PRG_Debug_View();

IF L_Run_Extended_Diagnostics THEN
    PRG_System_Diagnostics_Ext();
    GVL_MAIN_PHASE_FEEDBACK.G_Phase_08_Extended_Diagnostics_Executed := TRUE;
END_IF;

IF L_Run_Extended_Observability THEN
    PRG_System_History();
    PRG_System_BlackBox();
    PRG_System_Trend();
    GVL_MAIN_PHASE_FEEDBACK.G_Phase_08_Extended_Observability_Executed := TRUE;
END_IF;

IF L_Run_Simulation THEN
    PRG_System_Simulation();
    GVL_MAIN_PHASE_FEEDBACK.G_Phase_08_Simulation_Executed := TRUE;
END_IF;

GVL_MAIN_PHASE_FEEDBACK.G_Phase_08_Diagnostics_HMI_Executed := TRUE;
GVL_MAIN_PHASE_FEEDBACK.G_Phase_08_Diagnostics_HMI_Valid := TRUE;

IF L_Run_Extended_Diagnostics AND L_Run_Extended_Observability AND L_Run_Simulation THEN
    GVL_MAIN_PHASE_FEEDBACK.G_Phase_08_Diagnostics_HMI_Status_Text := 'Diagnostics/HMI phase executed';
ELSE
    GVL_MAIN_PHASE_FEEDBACK.G_Phase_08_Diagnostics_HMI_Status_Text := 'Diagnostics/HMI phase executed with designed shedding';
END_IF;

GVL_MAIN_PHASE_FEEDBACK.G_Critical_Path_Executed :=
    GVL_MAIN_PHASE_FEEDBACK.G_Phase_01_Bootstrap_Executed
    AND GVL_MAIN_PHASE_FEEDBACK.G_Phase_02_Redundancy_Executed
    AND GVL_MAIN_PHASE_FEEDBACK.G_Phase_03_Input_Safety_Command_Executed
    AND GVL_MAIN_PHASE_FEEDBACK.G_Phase_05_Domain_Output_Executed;

GVL_MAIN_PHASE_FEEDBACK.G_Critical_Path_Valid :=
    GVL_MAIN_PHASE_FEEDBACK.G_Phase_01_Bootstrap_Valid
    AND GVL_MAIN_PHASE_FEEDBACK.G_Phase_02_Redundancy_Valid
    AND GVL_MAIN_PHASE_FEEDBACK.G_Phase_03_Input_Safety_Command_Valid
    AND GVL_MAIN_PHASE_FEEDBACK.G_Phase_05_Domain_Output_Valid;

GVL_MAIN_PHASE_FEEDBACK.G_Observability_Path_Executed :=
    GVL_MAIN_PHASE_FEEDBACK.G_Phase_07_Semantic_Governance_Executed
    AND GVL_MAIN_PHASE_FEEDBACK.G_Phase_08_Diagnostics_HMI_Executed;

GVL_MAIN_PHASE_FEEDBACK.G_Observability_Path_Valid :=
    GVL_MAIN_PHASE_FEEDBACK.G_Phase_07_Semantic_Governance_Valid
    AND GVL_MAIN_PHASE_FEEDBACK.G_Phase_08_Diagnostics_HMI_Valid;

GVL_MAIN_PHASE_FEEDBACK.G_Any_Phase_Invalid :=
    NOT GVL_MAIN_PHASE_FEEDBACK.G_Phase_01_Bootstrap_Valid
    OR NOT GVL_MAIN_PHASE_FEEDBACK.G_Phase_02_Redundancy_Valid
    OR NOT GVL_MAIN_PHASE_FEEDBACK.G_Phase_03_Input_Safety_Command_Valid
    OR NOT GVL_MAIN_PHASE_FEEDBACK.G_Phase_04_Transport_Distributed_Valid
    OR NOT GVL_MAIN_PHASE_FEEDBACK.G_Phase_05_Domain_Output_Valid
    OR NOT GVL_MAIN_PHASE_FEEDBACK.G_Phase_06_PostOutput_Authority_Valid
    OR NOT GVL_MAIN_PHASE_FEEDBACK.G_Phase_07_Semantic_Governance_Valid
    OR NOT GVL_MAIN_PHASE_FEEDBACK.G_Phase_08_Diagnostics_HMI_Valid;

GVL_MAIN_PHASE_FEEDBACK.G_Any_Phase_Skipped_By_Design :=
    GVL_MAIN_PHASE_FEEDBACK.G_Phase_07_Full_Semantic_Skipped_By_Design
    OR GVL_MAIN_PHASE_FEEDBACK.G_Phase_07_Extended_Observability_Skipped_By_Design
    OR GVL_MAIN_PHASE_FEEDBACK.G_Phase_07_Analytics_Skipped_By_Design
    OR GVL_MAIN_PHASE_FEEDBACK.G_Phase_08_Extended_Diagnostics_Skipped_By_Design
    OR GVL_MAIN_PHASE_FEEDBACK.G_Phase_08_Extended_Observability_Skipped_By_Design
    OR GVL_MAIN_PHASE_FEEDBACK.G_Phase_08_Simulation_Skipped_By_Design;

IF GVL_MAIN_PHASE_FEEDBACK.G_Any_Phase_Invalid THEN
    GVL_MAIN_PHASE_FEEDBACK.G_Status_Code := 1;
    GVL_MAIN_PHASE_FEEDBACK.G_Status_Text := 'MAIN phase feedback degraded';
ELSIF GVL_MAIN_PHASE_FEEDBACK.G_Any_Phase_Skipped_By_Design THEN
    GVL_MAIN_PHASE_FEEDBACK.G_Status_Code := 2;
    GVL_MAIN_PHASE_FEEDBACK.G_Status_Text := 'MAIN phase feedback nominal with designed shedding';
ELSE
    GVL_MAIN_PHASE_FEEDBACK.G_Status_Code := 0;
    GVL_MAIN_PHASE_FEEDBACK.G_Status_Text := 'MAIN phase feedback nominal';
END_IF;

GVL_MAIN_PHASE_FEEDBACK.G_Current_Phase := 0;
GVL_MAIN_PHASE_FEEDBACK.G_Last_Update_MS := GVL_TIME_SERVICE.G_Now_MS;

// >>> BULK_SYNC_ANCHOR: PRG_Main_Phase_08_Diagnostics_HMI <<<
END_PROGRAM

(* ---- PRG_Modbus_Master.st ---- *)
PROGRAM PRG_Modbus_Master
VAR
    L_i : INT;
END_VAR

// ======================================================
// MODBUS MASTER RUNTIME SCHEDULER
// ======================================================
// This layer intentionally does not depend on a concrete
// CODESYS Modbus library.
//
// Future implementation options:
//   - CODESYS Modbus Serial Master RTU
//   - ModbusFB library
//   - Vendor-specific Modbus drivers
//
// Responsibilities:
//   1. Dispatch queued requests.
//   2. Apply timeout supervision.
//   3. Publish response state.
//   4. Protect transport execution ordering.
//
// Safety rule:
//   Until a concrete Modbus RTU driver is wired here, this PRG must NOT
//   produce fake successful responses.
// ======================================================

IF NOT GVL_CONFIG.G_OpenTherm_Enabled THEN
    GVL_MODBUS_MASTER.G_Master_Online := FALSE;
    GVL_MODBUS_MASTER.G_Master_Error := FALSE;

    FOR L_i := 1 TO 16 DO
        GVL_MODBUS_MASTER.G_Response[L_i].Busy := FALSE;
        GVL_MODBUS_MASTER.G_Response[L_i].Done := FALSE;
        GVL_MODBUS_MASTER.G_Response[L_i].Error := FALSE;
        GVL_MODBUS_MASTER.G_Response[L_i].Error_Code := 0;
    END_FOR;

    RETURN;
END_IF;

// No concrete RTU/TCP implementation is attached yet.
// Keep the master offline instead of simulating a response.
GVL_MODBUS_MASTER.G_Master_Online := FALSE;
GVL_MODBUS_MASTER.G_Master_Error := TRUE;

FOR L_i := 1 TO 16 DO

    IF GVL_MODBUS_MASTER.G_Request[L_i].Enable THEN
        GVL_MODBUS_MASTER.G_Response[L_i].Busy := FALSE;
        GVL_MODBUS_MASTER.G_Response[L_i].Done := FALSE;
        GVL_MODBUS_MASTER.G_Response[L_i].Error := TRUE;
        GVL_MODBUS_MASTER.G_Response[L_i].Error_Code := 16#0001;
        GVL_MODBUS_MASTER.G_Response[L_i].Last_Sequence :=
            GVL_MODBUS_MASTER.G_Request[L_i].Sequence;
        GVL_MODBUS_MASTER.G_Response[L_i].Last_Update_MS :=
            GVL_STATUS.G_System_Time_MS;
    ELSE
        GVL_MODBUS_MASTER.G_Response[L_i].Busy := FALSE;
        GVL_MODBUS_MASTER.G_Response[L_i].Done := FALSE;
    END_IF;

END_FOR;

END_PROGRAM

(* ---- PRG_Modbus_RTU_Driver.st ---- *)
PROGRAM PRG_Modbus_RTU_Driver
VAR
    FB_RTU_Driver : FB_Modbus_RTU_Driver;
END_VAR

// ======================================================
// MODBUS RTU DRIVER EXECUTION
// ======================================================
// Runtime execution wrapper for the RTU driver FB.
//
// Driver_Attached is a configuration/HMI decision and must not depend
// on runtime bridge state.
// ======================================================

FB_RTU_Driver(
    VI_Enable := GVL_CONFIG.G_OpenTherm_Enabled,
    VI_Driver_Attached := GVL_CONFIG.G_Modbus_RTU_Driver_Attached,
    VI_System_Time_MS := GVL_STATUS.G_System_Time_MS
);

END_PROGRAM

(* ---- PRG_Modbus_RTU_SysCom_Backend.st ---- *)
PROGRAM PRG_Modbus_RTU_SysCom_Backend
VAR
    FB_Backend : FB_Modbus_RTU_SysCom_Backend;
END_VAR

FB_Backend(
    VI_Enable := GVL_CONFIG.G_OpenTherm_Enabled,
    VI_System_Time_MS := GVL_STATUS.G_System_Time_MS
);

END_PROGRAM

(* ---- PRG_Mode_Manager.st ---- *)
PROGRAM PRG_Mode_Manager
VAR
    fbMode : FB_Mode_Manager;
    L_Last_Mode : E_Behavior_Mode := BEHAVIOR_HOME;
END_VAR

fbMode(
    VI_Is_Night := GVL_STATUS.G_Is_Night,
    VI_System_Time_MS := GVL_STATUS.G_System_Time_MS
);

GVL_MODE.G_Current_Behavior_Mode := fbMode.VO_Mode;
GVL_MODE.G_Mode_Code := fbMode.VO_Mode_Code;

IF L_Last_Mode <> fbMode.VO_Mode THEN
    GVL_MODE.G_Mode_Last_Change_TS := GVL_STATUS.G_System_Time_MS;
    L_Last_Mode := fbMode.VO_Mode;
END_IF;

(* ---- PRG_Observability_Governor.st ---- *)
PROGRAM PRG_Observability_Governor
VAR
    L_Now_MS : UDINT;

    L_Runtime_Authority_Valid : BOOL;
    L_Publication_Authority_Valid : BOOL;
    L_Recovery_Authority_Valid : BOOL;
    L_Distributed_Authority_Valid : BOOL;
    L_Final_Projection_Barrier_Valid : BOOL;
END_VAR

L_Now_MS := GVL_STATUS.G_System_Time_MS;

GVL_OBSERVABILITY_AUTHORITY.Runtime_Failure_Visible := FALSE;
GVL_OBSERVABILITY_AUTHORITY.Output_Decay_Visible := FALSE;
GVL_OBSERVABILITY_AUTHORITY.Transport_Failure_Visible := FALSE;
GVL_OBSERVABILITY_AUTHORITY.Recovery_Failure_Visible := FALSE;
GVL_OBSERVABILITY_AUTHORITY.Fencing_Failure_Visible := FALSE;
GVL_OBSERVABILITY_AUTHORITY.Monotonic_Failure_Visible := FALSE;

GVL_OBSERVABILITY_AUTHORITY.Distributed_Failure_Visible := FALSE;
GVL_OBSERVABILITY_AUTHORITY.Distributed_Quarantine_Visible := FALSE;
GVL_OBSERVABILITY_AUTHORITY.Peer_Runtime_Stale_Visible := FALSE;
GVL_OBSERVABILITY_AUTHORITY.Peer_Snapshot_Stale_Visible := FALSE;
GVL_OBSERVABILITY_AUTHORITY.Peer_Boot_Mismatch_Visible := FALSE;
GVL_OBSERVABILITY_AUTHORITY.Peer_Fencing_Conflict_Visible := FALSE;
GVL_OBSERVABILITY_AUTHORITY.Peer_Semantic_Continuity_Lost_Visible := FALSE;

GVL_OBSERVABILITY_AUTHORITY.Distributed_Publication_Reconciliation_Visible := FALSE;
GVL_OBSERVABILITY_AUTHORITY.Distributed_Publication_Freeze_Visible := FALSE;
GVL_OBSERVABILITY_AUTHORITY.Distributed_Snapshot_Consistency_Visible := FALSE;
GVL_OBSERVABILITY_AUTHORITY.Peer_Publication_Stale_Visible := FALSE;
GVL_OBSERVABILITY_AUTHORITY.Peer_Publication_Divergence_Visible := FALSE;
GVL_OBSERVABILITY_AUTHORITY.Peer_Publication_Reconciliation_Lost_Visible := FALSE;
GVL_OBSERVABILITY_AUTHORITY.Peer_Snapshot_Not_Immutable_Visible := FALSE;
GVL_OBSERVABILITY_AUTHORITY.Distributed_Immutable_Snapshot_Quarantine_Visible := FALSE;

GVL_OBSERVABILITY_AUTHORITY.Distributed_Commit_Visible := FALSE;
GVL_OBSERVABILITY_AUTHORITY.Distributed_Commit_Quarantine_Visible := FALSE;
GVL_OBSERVABILITY_AUTHORITY.Publication_Prepare_Visible := FALSE;
GVL_OBSERVABILITY_AUTHORITY.Publication_Commit_Visible := FALSE;
GVL_OBSERVABILITY_AUTHORITY.Peer_Commit_Ack_Visible := FALSE;
GVL_OBSERVABILITY_AUTHORITY.Peer_Commit_Mismatch_Visible := FALSE;
GVL_OBSERVABILITY_AUTHORITY.Peer_Commit_Replay_Visible := FALSE;
GVL_OBSERVABILITY_AUTHORITY.Peer_Commit_Missing_Visible := FALSE;
GVL_OBSERVABILITY_AUTHORITY.Commit_Lease_Expired_Visible := FALSE;

GVL_OBSERVABILITY_AUTHORITY.Unsafe_State_Published := FALSE;
GVL_OBSERVABILITY_AUTHORITY.Emergency_Visibility_Required := FALSE;

L_Runtime_Authority_Valid :=
    GVL_RUNTIME_EPOCH.Runtime_Runtime_Barrier_OK
    AND GVL_RUNTIME_SNAPSHOT.Snapshot_Publication_Allowed
    AND GVL_RUNTIME_SNAPSHOT.Snapshot_Copy_Valid
    AND GVL_RUNTIME_SNAPSHOT.Snapshot_Isolation_Valid
    AND NOT GVL_RUNTIME_SNAPSHOT.Snapshot_Mutation_Detected;

L_Publication_Authority_Valid :=
    GVL_OUTPUT_EPOCH.Output_Publication_Allowed
    AND GVL_OUTPUT_EPOCH.Output_Publication_Valid
    AND GVL_OUTPUT_EPOCH.Output_Runtime_Epoch_Valid
    AND NOT GVL_OUTPUT_EPOCH.Output_Lease_Expired
    AND NOT GVL_OUTPUT_EPOCH.Output_Forced_Safe_Decay
    AND GVL_TRANSPORT_FRESHNESS.Transport_Freshness_Valid;

L_Recovery_Authority_Valid :=
    GVL_RECOVERY_GOVERNANCE.Recovery_Governance_Valid
    AND NOT GVL_RECOVERY_GOVERNANCE.Recovery_Quarantine_Active
    AND GVL_CONVERGENCE.Convergence_Release_Allowed;

L_Distributed_Authority_Valid :=
    GVL_DISTRIBUTED_EPOCH.Distributed_Reconciliation_Valid
    AND NOT GVL_DISTRIBUTED_EPOCH.Distributed_Quarantine_Active
    AND GVL_DISTRIBUTED_SNAPSHOT.Distributed_Snapshot_Consistent
    AND GVL_DISTRIBUTED_COMMIT.Distributed_Commit_Valid
    AND GVL_Distributed_Execution_Gates.G_Runtime_Valid;

// Final projection proof barrier.
L_Final_Projection_Barrier_Valid :=
    GVL_COMMAND_VERIFY.PreOutput_Barrier_OK
    AND NOT GVL_COMMAND_VERIFY.PreOutput_Block_IO;

GVL_OBSERVABILITY_AUTHORITY.Publication_Runtime_Valid :=
    L_Runtime_Authority_Valid
    AND L_Publication_Authority_Valid
    AND L_Recovery_Authority_Valid
    AND L_Distributed_Authority_Valid
    AND L_Final_Projection_Barrier_Valid;

IF NOT L_Final_Projection_Barrier_Valid THEN
    GVL_OBSERVABILITY_AUTHORITY.Unsafe_State_Published := TRUE;
    GVL_OBSERVABILITY_AUTHORITY.Emergency_Visibility_Required := TRUE;
END_IF;

IF NOT L_Publication_Authority_Valid THEN
    GVL_OBSERVABILITY_AUTHORITY.Output_Decay_Visible := TRUE;
    GVL_OBSERVABILITY_AUTHORITY.Emergency_Visibility_Required := TRUE;
END_IF;

GVL_OBSERVABILITY_AUTHORITY.Observability_Epoch := GVL_OBSERVABILITY_AUTHORITY.Observability_Epoch + 1;
GVL_OBSERVABILITY_AUTHORITY.Observability_Snapshot_Epoch := GVL_OBSERVABILITY_AUTHORITY.Observability_Snapshot_Epoch + 1;

GVL_OBSERVABILITY_AUTHORITY.Observability_Last_Publication_MS := L_Now_MS;

GVL_OBSERVABILITY_AUTHORITY.Observability_Last_Error_Code := 0;
GVL_OBSERVABILITY_AUTHORITY.Observability_Last_Error_Text := '';
END_PROGRAM

(* ---- PRG_Observability_Truth_Governor.st ---- *)
PROGRAM PRG_Observability_Truth_Governor
VAR
    L_Now_MS : UDINT;
    L_Observability_Valid : BOOL := TRUE;
    L_Error_Code : UDINT := 0;
    L_Error_Text : STRING(160) := '';
END_VAR

L_Now_MS := GVL_STATUS.G_System_Time_MS;
L_Observability_Valid := TRUE;
L_Error_Code := 0;
L_Error_Text := '';

// Fail-safe defaults.
GVL_OBSERVABILITY_TRUTH.Observability_Truth_Valid := FALSE;
GVL_OBSERVABILITY_TRUTH.Observability_Truth_Granted := FALSE;
GVL_OBSERVABILITY_TRUTH.Observability_Truth_Quarantine_Active := TRUE;

GVL_OBSERVABILITY_TRUTH.HMI_Authority_Coherent := FALSE;
GVL_OBSERVABILITY_TRUTH.Alarm_Authority_Coherent := FALSE;
GVL_OBSERVABILITY_TRUTH.Trend_Authority_Coherent := FALSE;
GVL_OBSERVABILITY_TRUTH.Diagnostics_Authority_Coherent := FALSE;
GVL_OBSERVABILITY_TRUTH.History_Authority_Coherent := FALSE;

// Semantic continuity authority required.
IF NOT GVL_SEMANTIC_CONTINUITY.Semantic_Continuity_Granted THEN
    L_Observability_Valid := FALSE;
    L_Error_Code := 32000;
    L_Error_Text := 'Semantic continuity authority not granted';
END_IF;

// Observability split-brain detectors.
IF GVL_OBSERVABILITY_TRUTH.Stale_HMI_Epoch_Detected THEN
    L_Observability_Valid := FALSE;
    L_Error_Code := 32001;
    L_Error_Text := 'Stale HMI epoch detected';
END_IF;

IF GVL_OBSERVABILITY_TRUTH.Alarm_Publication_Lag_Detected THEN
    L_Observability_Valid := FALSE;
    L_Error_Code := 32002;
    L_Error_Text := 'Alarm publication lag detected';
END_IF;

IF GVL_OBSERVABILITY_TRUTH.Trend_Causality_Skew_Detected THEN
    L_Observability_Valid := FALSE;
    L_Error_Code := 32003;
    L_Error_Text := 'Trend causality skew detected';
END_IF;

IF GVL_OBSERVABILITY_TRUTH.Diagnostic_Truth_Race_Detected THEN
    L_Observability_Valid := FALSE;
    L_Error_Code := 32004;
    L_Error_Text := 'Diagnostic truth race detected';
END_IF;

IF GVL_OBSERVABILITY_TRUTH.Operator_Visibility_Fragmentation_Detected THEN
    L_Observability_Valid := FALSE;
    L_Error_Code := 32005;
    L_Error_Text := 'Operator visibility fragmentation detected';
END_IF;

IF GVL_OBSERVABILITY_TRUTH.Authority_UI_Divergence_Detected THEN
    L_Observability_Valid := FALSE;
    L_Error_Code := 32006;
    L_Error_Text := 'Authority/UI divergence detected';
END_IF;

// Projection causality validation.
IF L_Observability_Valid
AND NOT GVL_OBSERVABILITY_TRUTH.HMI_Epoch_Coherent THEN
    L_Observability_Valid := FALSE;
    L_Error_Code := 32010;
    L_Error_Text := 'HMI epoch coherence invalid';
END_IF;

IF L_Observability_Valid
AND NOT GVL_OBSERVABILITY_TRUTH.Alarm_Publication_Coherent THEN
    L_Observability_Valid := FALSE;
    L_Error_Code := 32011;
    L_Error_Text := 'Alarm publication coherence invalid';
END_IF;

IF L_Observability_Valid
AND NOT GVL_OBSERVABILITY_TRUTH.Trend_Causality_Coherent THEN
    L_Observability_Valid := FALSE;
    L_Error_Code := 32012;
    L_Error_Text := 'Trend causality coherence invalid';
END_IF;

IF L_Observability_Valid
AND NOT GVL_OBSERVABILITY_TRUTH.Diagnostics_Causality_Coherent THEN
    L_Observability_Valid := FALSE;
    L_Error_Code := 32013;
    L_Error_Text := 'Diagnostics causality coherence invalid';
END_IF;

IF L_Observability_Valid
AND NOT GVL_OBSERVABILITY_TRUTH.Operator_Visibility_Consistent THEN
    L_Observability_Valid := FALSE;
    L_Error_Code := 32014;
    L_Error_Text := 'Operator visibility consistency invalid';
END_IF;

IF L_Observability_Valid THEN
    GVL_OBSERVABILITY_TRUTH.Observability_Truth_Valid := TRUE;
    GVL_OBSERVABILITY_TRUTH.Observability_Truth_Granted := TRUE;
    GVL_OBSERVABILITY_TRUTH.Observability_Truth_Quarantine_Active := FALSE;

    GVL_OBSERVABILITY_TRUTH.HMI_Authority_Coherent := TRUE;
    GVL_OBSERVABILITY_TRUTH.Alarm_Authority_Coherent := TRUE;
    GVL_OBSERVABILITY_TRUTH.Trend_Authority_Coherent := TRUE;
    GVL_OBSERVABILITY_TRUTH.Diagnostics_Authority_Coherent := TRUE;
    GVL_OBSERVABILITY_TRUTH.History_Authority_Coherent := TRUE;

    GVL_OBSERVABILITY_TRUTH.Observability_Truth_Epoch :=
        GVL_SEMANTIC_CONTINUITY.Semantic_Continuity_Epoch;

    GVL_OBSERVABILITY_TRUTH.Observability_Truth_Epoch_Coherent := TRUE;

    GVL_OBSERVABILITY_TRUTH.Observability_Last_Update_MS := L_Now_MS;
    GVL_OBSERVABILITY_TRUTH.Observability_Lease_Expired := FALSE;

    GVL_OBSERVABILITY_TRUTH.Observability_Last_Error_Code := 0;
    GVL_OBSERVABILITY_TRUTH.Observability_Last_Error_Text := '';
ELSE
    GVL_OBSERVABILITY_TRUTH.Observability_Truth_Valid := FALSE;
    GVL_OBSERVABILITY_TRUTH.Observability_Truth_Granted := FALSE;
    GVL_OBSERVABILITY_TRUTH.Observability_Truth_Quarantine_Active := TRUE;

    GVL_OBSERVABILITY_TRUTH.Observability_Lease_Expired := TRUE;

    GVL_OBSERVABILITY_TRUTH.Observability_Last_Error_Code :=
        L_Error_Code;

    GVL_OBSERVABILITY_TRUTH.Observability_Last_Error_Text :=
        L_Error_Text;

    GVL_OBSERVABILITY_TRUTH.Observability_Invalidation_Count :=
        GVL_OBSERVABILITY_TRUTH.Observability_Invalidation_Count + 1;
END_IF;

END_PROGRAM

(* ---- PRG_OpenTherm_Adapter_Status.st ---- *)
PROGRAM PRG_OpenTherm_Adapter_Status
VAR
    L_i : INT;
    L_Now_MS : UDINT;
    L_Heartbeat_Age : UDINT;
    L_Command_Age : UDINT;
END_VAR

L_Now_MS := GVL_STATUS.G_System_Time_MS;

FOR L_i := 1 TO GVL_CONSTANTS.C_MAX_BOILERS DO

    // ======================================================
    // HEARTBEAT VALIDATION
    // ======================================================
    IF GVL_OPENTHERM_ADAPTER.G_Status[L_i].Raw_Heartbeat <>
       GVL_OPENTHERM_ADAPTER.G_Status[L_i].Last_Heartbeat THEN

        GVL_OPENTHERM_ADAPTER.G_Status[L_i].Last_Heartbeat :=
            GVL_OPENTHERM_ADAPTER.G_Status[L_i].Raw_Heartbeat;

        GVL_OPENTHERM_ADAPTER.G_Status[L_i].Last_Heartbeat_MS := L_Now_MS;
    END_IF;

    L_Heartbeat_Age :=
        L_Now_MS - GVL_OPENTHERM_ADAPTER.G_Status[L_i].Last_Heartbeat_MS;

    GVL_OPENTHERM_ADAPTER.G_Status[L_i].Heartbeat_Age_MS :=
        L_Heartbeat_Age;

    GVL_OPENTHERM_ADAPTER.G_Status[L_i].Heartbeat_Timeout :=
        (L_Heartbeat_Age > GVL_CONFIG.G_OpenTherm_Heartbeat_Timeout_MS);

    // ======================================================
    // COMMAND ACK VALIDATION
    // ======================================================
    GVL_OPENTHERM_ADAPTER.G_Status[L_i].Command_Ack :=
        (GVL_OPENTHERM_ADAPTER.G_Status[L_i].Raw_Ack_Seq =
         GVL_OPENTHERM_ADAPTER.G_Command[L_i].Sequence);

    GVL_OPENTHERM_ADAPTER.G_Status[L_i].Last_Command_Ack_Seq :=
        GVL_OPENTHERM_ADAPTER.G_Status[L_i].Raw_Ack_Seq;

    L_Command_Age :=
        L_Now_MS - GVL_OPENTHERM_ADAPTER.G_Command[L_i].Last_Write_MS;

    GVL_OPENTHERM_ADAPTER.G_Status[L_i].Command_Age_MS :=
        L_Command_Age;

    GVL_OPENTHERM_ADAPTER.G_Status[L_i].Command_Timeout :=
        (NOT GVL_OPENTHERM_ADAPTER.G_Status[L_i].Command_Ack) AND
        (L_Command_Age > GVL_CONFIG.G_OpenTherm_Command_Ack_Timeout_MS);

    // ======================================================
    // FINAL ADAPTER STATE
    // ======================================================
    GVL_OPENTHERM_ADAPTER.G_Status[L_i].Adapter_Online :=
        GVL_OPENTHERM_ADAPTER.G_Status[L_i].Raw_Online AND
        (NOT GVL_OPENTHERM_ADAPTER.G_Status[L_i].Heartbeat_Timeout) AND
        (NOT GVL_OPENTHERM_ADAPTER.G_Status[L_i].Command_Timeout);

    GVL_OPENTHERM_ADAPTER.G_Status[L_i].Adapter_Error :=
        GVL_OPENTHERM_ADAPTER.G_Status[L_i].Raw_Error OR
        GVL_OPENTHERM_ADAPTER.G_Status[L_i].Command_Timeout OR
        GVL_OPENTHERM_ADAPTER.G_Status[L_i].Heartbeat_Timeout;

    // ======================================================
    // ENUM STATES
    // ======================================================
    IF GVL_OPENTHERM_ADAPTER.G_Status[L_i].Heartbeat_Timeout THEN
        GVL_OPENTHERM_ADAPTER.G_Status[L_i].Adapter_State := OT_STATE_HEARTBEAT_TIMEOUT;
        GVL_OPENTHERM_ADAPTER.G_Status[L_i].Error_State := OT_ERROR_HEARTBEAT_TIMEOUT;

    ELSIF GVL_OPENTHERM_ADAPTER.G_Status[L_i].Command_Timeout THEN
        GVL_OPENTHERM_ADAPTER.G_Status[L_i].Adapter_State := OT_STATE_ACK_TIMEOUT;
        GVL_OPENTHERM_ADAPTER.G_Status[L_i].Error_State := OT_ERROR_ACK_TIMEOUT;

    ELSIF GVL_OPENTHERM_ADAPTER.G_Status[L_i].Raw_Error THEN
        GVL_OPENTHERM_ADAPTER.G_Status[L_i].Adapter_State := OT_STATE_ADAPTER_ERROR;
        GVL_OPENTHERM_ADAPTER.G_Status[L_i].Error_State := OT_ERROR_ADAPTER_FAULT;

    ELSIF GVL_OPENTHERM_ADAPTER.G_Status[L_i].Adapter_Online THEN
        GVL_OPENTHERM_ADAPTER.G_Status[L_i].Adapter_State := OT_STATE_ONLINE;
        GVL_OPENTHERM_ADAPTER.G_Status[L_i].Error_State := OT_ERROR_NONE;

    ELSE
        GVL_OPENTHERM_ADAPTER.G_Status[L_i].Adapter_State := OT_STATE_OFFLINE;
        GVL_OPENTHERM_ADAPTER.G_Status[L_i].Error_State := OT_ERROR_COMMUNICATION;
    END_IF;

    // ======================================================
    // PUBLISH TO SYSTEM STATE
    // ======================================================
    GVL_STATE.G_Boiler_OT_Online[L_i] :=
        GVL_OPENTHERM_ADAPTER.G_Status[L_i].Adapter_Online;

    GVL_STATE.G_Boiler_OT_Command_Ack[L_i] :=
        GVL_OPENTHERM_ADAPTER.G_Status[L_i].Command_Ack;

    GVL_STATE.G_Boiler_OT_Command_Timeout[L_i] :=
        GVL_OPENTHERM_ADAPTER.G_Status[L_i].Command_Timeout;

    GVL_STATE.G_Boiler_OT_Heartbeat_Timeout[L_i] :=
        GVL_OPENTHERM_ADAPTER.G_Status[L_i].Heartbeat_Timeout;

    GVL_STATE.G_Boiler_OT_Adapter_Error[L_i] :=
        GVL_OPENTHERM_ADAPTER.G_Status[L_i].Adapter_Error;

    GVL_STATE.G_Boiler_OT_Heartbeat_Age_MS[L_i] :=
        GVL_OPENTHERM_ADAPTER.G_Status[L_i].Heartbeat_Age_MS;

    GVL_STATE.G_Boiler_OT_Command_Age_MS[L_i] :=
        GVL_OPENTHERM_ADAPTER.G_Status[L_i].Command_Age_MS;

    GVL_STATE.G_Boiler_Error[L_i] :=
        GVL_OPENTHERM_ADAPTER.G_Status[L_i].Adapter_Error;

    GVL_STATE.G_Boiler_Flame[L_i] :=
        GVL_OPENTHERM_ADAPTER.G_Status[L_i].Raw_Flame;

END_FOR;

END_PROGRAM

(* ---- PRG_OpenTherm_Command_Interface.st ---- *)
PROGRAM PRG_OpenTherm_Command_Interface
VAR
    fbBoilerOpenThermInterface : FB_Boiler_OpenTherm_Interface;
    L_i : INT;
    L_Enable : ARRAY[1..GVL_CONSTANTS.C_MAX_BOILERS] OF BOOL;
    L_Setpoint : ARRAY[1..GVL_CONSTANTS.C_MAX_BOILERS] OF REAL;
    L_Safety_Stop : BOOL;
END_VAR

L_Safety_Stop :=
    GVL_COMMAND_SHADOW.G_Boiler_Stop OR
    GVL_COMMAND_SHADOW.G_Heating_Gas_Safety_Stop OR
    (GVL_SAFETY_SHUTDOWN.G_Safety_Mode = GAS) OR
    (GVL_SAFETY_SHUTDOWN.G_Safety_Mode = GLOBAL_STOP);

FOR L_i := 1 TO GVL_CONSTANTS.C_MAX_BOILERS DO
    IF L_Safety_Stop THEN
        L_Enable[L_i] := FALSE;
        L_Setpoint[L_i] := 0.0;
    ELSE
        L_Enable[L_i] := GVL_STATE.G_Boiler_OT_Enable[L_i];
        L_Setpoint[L_i] := GVL_STATE.G_Boiler_OT_Setpoint[L_i];
    END_IF;
END_FOR;

fbBoilerOpenThermInterface(
    VI_Enable := L_Enable,
    VI_Setpoint := L_Setpoint,
    VI_OT_Online := GVL_STATE.G_Boiler_OT_Online,
    VI_OT_Error := GVL_STATE.G_Boiler_OT_Adapter_Error
);

FOR L_i := 1 TO GVL_CONSTANTS.C_MAX_BOILERS DO
    GVL_STATE.G_Boiler_OT_Enable[L_i] := fbBoilerOpenThermInterface.VO_OT_Enable[L_i];
    GVL_STATE.G_Boiler_OT_Setpoint[L_i] := fbBoilerOpenThermInterface.VO_OT_Setpoint[L_i];
    GVL_STATE.G_Boiler_OT_Command_Ack[L_i] := fbBoilerOpenThermInterface.VO_OT_Command_Valid[L_i];
END_FOR;

// >>> BULK_SYNC_ANCHOR: PRG_OpenTherm_Command_Interface <<<
END_PROGRAM

(* ---- PRG_OpenTherm_Transport.st ---- *)
PROGRAM PRG_OpenTherm_Transport
VAR
    L_i : INT;
    L_Status_Word : WORD;
    L_Heartbeat : UDINT;
    L_Ack_Seq : UDINT;
END_VAR

// ======================================================
// REAL TRANSPORT LAYER CONTRACT
// ======================================================
// This layer converts high-level command/status structures
// into transport-safe wire images.
//
// Real Modbus RTU/TCP or serial IO code must:
//   1. Write G_Wire_Image command fields to adapter registers.
//   2. Read adapter status registers into G_Wire_Image status fields.
//
// This program keeps all protocol decoding centralized.
// ======================================================

GVL_OPENTHERM_ADAPTER.G_Transport_Online := TRUE;
GVL_OPENTHERM_ADAPTER.G_Transport_Error := FALSE;
GVL_OPENTHERM_ADAPTER.G_Last_Transport_Update_MS := GVL_STATUS.G_System_Time_MS;

FOR L_i := 1 TO GVL_CONSTANTS.C_MAX_BOILERS DO

    // ======================================================
    // COMMAND → WIRE IMAGE
    // ======================================================
    IF GVL_OPENTHERM_ADAPTER.G_Command[L_i].Enable THEN
        GVL_OPENTHERM_ADAPTER.G_Wire_Image[L_i].Cmd_Enable := 1;
    ELSE
        GVL_OPENTHERM_ADAPTER.G_Wire_Image[L_i].Cmd_Enable := 0;
    END_IF;

    GVL_OPENTHERM_ADAPTER.G_Wire_Image[L_i].Cmd_Setpoint_x10 :=
        GVL_OPENTHERM_ADAPTER.G_Command[L_i].Setpoint_x10;

    GVL_OPENTHERM_ADAPTER.G_Wire_Image[L_i].Cmd_Seq_Lo :=
        UDINT_TO_WORD(GVL_OPENTHERM_ADAPTER.G_Command[L_i].Sequence AND 16#FFFF);

    GVL_OPENTHERM_ADAPTER.G_Wire_Image[L_i].Cmd_Seq_Hi :=
        UDINT_TO_WORD(SHR(GVL_OPENTHERM_ADAPTER.G_Command[L_i].Sequence, 16));

    // ======================================================
    // WIRE IMAGE → STATUS
    // ======================================================
    L_Heartbeat :=
        WORD_TO_UDINT(GVL_OPENTHERM_ADAPTER.G_Wire_Image[L_i].Status_Heartbeat_Lo)
        OR SHL(
            WORD_TO_UDINT(GVL_OPENTHERM_ADAPTER.G_Wire_Image[L_i].Status_Heartbeat_Hi),
            16
        );

    L_Ack_Seq :=
        WORD_TO_UDINT(GVL_OPENTHERM_ADAPTER.G_Wire_Image[L_i].Status_Ack_Seq_Lo)
        OR SHL(
            WORD_TO_UDINT(GVL_OPENTHERM_ADAPTER.G_Wire_Image[L_i].Status_Ack_Seq_Hi),
            16
        );

    GVL_OPENTHERM_ADAPTER.G_Status[L_i].Raw_Heartbeat := L_Heartbeat;
    GVL_OPENTHERM_ADAPTER.G_Status[L_i].Raw_Ack_Seq := L_Ack_Seq;

    L_Status_Word :=
        GVL_OPENTHERM_ADAPTER.G_Wire_Image[L_i].Status_Word;

    GVL_OPENTHERM_ADAPTER.G_Status[L_i].Raw_Online :=
        (L_Status_Word AND 16#0001) <> 0;

    GVL_OPENTHERM_ADAPTER.G_Status[L_i].Raw_Error :=
        (L_Status_Word AND 16#0002) <> 0;

    GVL_OPENTHERM_ADAPTER.G_Status[L_i].Raw_Flame :=
        (L_Status_Word AND 16#0004) <> 0;

    GVL_OPENTHERM_ADAPTER.G_Status[L_i].Raw_Status_Word :=
        L_Status_Word;

    GVL_OPENTHERM_ADAPTER.G_Status[L_i].Raw_Error_Code :=
        GVL_OPENTHERM_ADAPTER.G_Wire_Image[L_i].Error_Code;

    GVL_OPENTHERM_ADAPTER.G_Status[L_i].Raw_Modulation_x10 :=
        GVL_OPENTHERM_ADAPTER.G_Wire_Image[L_i].Modulation_x10;

    GVL_OPENTHERM_ADAPTER.G_Status[L_i].Raw_Boiler_Temp_x10 :=
        WORD_TO_INT(GVL_OPENTHERM_ADAPTER.G_Wire_Image[L_i].Boiler_Temp_x10);

END_FOR;

END_PROGRAM
